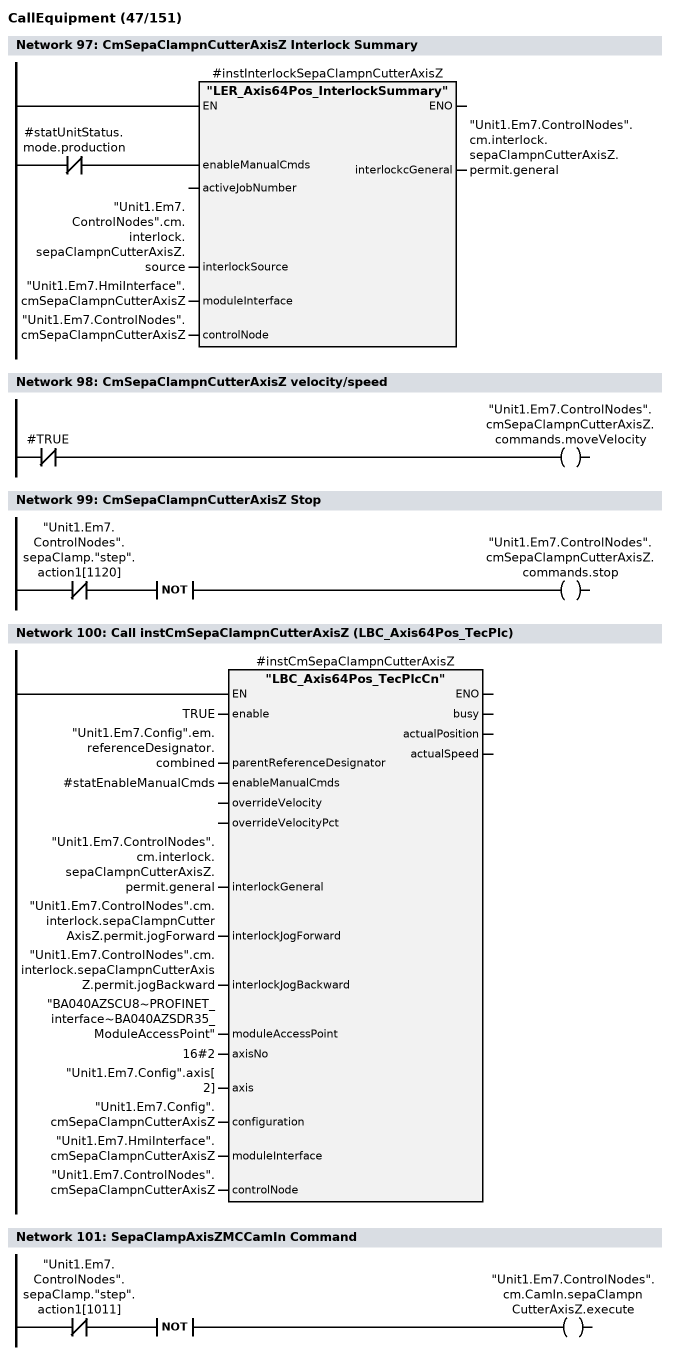
   RUNG wire#powerrail
      #instInterlockSepaClampnCutterAxisZ(enableManualCmds := wire#w1, activeJobNumber :=, interlockSource := "Unit1.Em7.ControlNodes".cm.interlock.sepaClampnCutterAxisZ.source, moduleInterface := "Unit1.Em7.HmiInterface".cmSepaClampnCutterAxisZ, controlNode := "Unit1.Em7.ControlNodes".cmSepaClampnCutterAxisZ, interlockcGeneral => "Unit1.Em7.ControlNodes".cm.interlock.sepaClampnCutterAxisZ.permit.general)
   END_RUNG
   RUNG wire#powerrail
      I_Contact( #statUnitStatus.mode.production )
   END_RUNG wire#w1
   // the same network as SCL:
   #instInterlockSepaClampnCutterAxisZ(enableManualCmds := NOT #statUnitStatus.mode.production,   // "LER_Axis64Pos_InterlockSummary"
                           interlockSource := "Unit1.Em7.ControlNodes".cm.interlock.sepaClampnCutterAxisZ.source,
                           moduleInterface := "Unit1.Em7.HmiInterface".cmSepaClampnCutterAxisZ,
                           controlNode := "Unit1.Em7.ControlNodes".cmSepaClampnCutterAxisZ,
                           interlockcGeneral => "Unit1.Em7.ControlNodes".cm.interlock.sepaClampnCutterAxisZ.permit.general);
END_REGION

REGION Network 98: CmSepaClampnCutterAxisZ velocity/speed
   RUNG wire#powerrail
      I_Contact( #TRUE )
      Coil( "Unit1.Em7.ControlNodes".cmSepaClampnCutterAxisZ.commands.moveVelocity )
   END_RUNG
   // the same network as SCL:
   "Unit1.Em7.ControlNodes".cmSepaClampnCutterAxisZ.commands.moveVelocity := NOT #TRUE;
END_REGION

REGION Network 99: CmSepaClampnCutterAxisZ Stop
   RUNG wire#powerrail
      I_Contact( "Unit1.Em7.ControlNodes".sepaClamp."step".action1[1120] )
      Not()
      Coil( "Unit1.Em7.ControlNodes".cmSepaClampnCutterAxisZ.commands.stop )
   END_RUNG
   // the same network as SCL:
   "Unit1.Em7.ControlNodes".cmSepaClampnCutterAxisZ.commands.stop := NOT (NOT "Unit1.Em7.ControlNodes".sepaClamp."step".action1[1120]);
END_REGION

REGION Network 100: Call instCmSepaClampnCutterAxisZ (LBC_Axis64Pos_TecPlc)
   RUNG wire#powerrail
      #instCmSepaClampnCutterAxisZ(enable := TRUE, parentReferenceDesignator := "Unit1.Em7.Config".em.referenceDesignator.combined, enableManualCmds := #statEnableManualCmds, overrideVelocity :=, overrideVelocityPct :=, interlockGeneral := "Unit1.Em7.ControlNodes".cm.interlock.sepaClampnCutterAxisZ.permit.general, interlockJogForward := "Unit1.Em7.ControlNodes".cm.interlock.sepaClampnCutterAxisZ.permit.jogForward, interlockJogBackward := "Unit1.Em7.ControlNodes".cm.interlock.sepaClampnCutterAxisZ.permit.jogBackward, moduleAccessPoint := "BA040AZSCU8~PROFINET_interface~BA040AZSDR35_ModuleAccessPoint", axisNo := 16#2, axis := "Unit1.Em7.Config".axis[2], configuration := "Unit1.Em7.Config".cmSepaClampnCutterAxisZ, moduleInterface := "Unit1.Em7.HmiInterface".cmSepaClampnCutterAxisZ, controlNode := "Unit1.Em7.ControlNodes".cmSepaClampnCutterAxisZ, busy =>, actualPosition =>, actualSpeed =>)
   END_RUNG
   // the same network as SCL:
   #instCmSepaClampnCutterAxisZ(enable := TRUE,   // "LBC_Axis64Pos_TecPlcCn"
                           parentReferenceDesignator := "Unit1.Em7.Config".em.referenceDesignator.combined,
                           enableManualCmds := #statEnableManualCmds,
                           interlockGeneral := "Unit1.Em7.ControlNodes".cm.interlock.sepaClampnCutterAxisZ.permit.general,
                           interlockJogForward := "Unit1.Em7.ControlNodes".cm.interlock.sepaClampnCutterAxisZ.permit.jogForward,
                           interlockJogBackward := "Unit1.Em7.ControlNodes".cm.interlock.sepaClampnCutterAxisZ.permit.jogBackward,
                           moduleAccessPoint := "BA040AZSCU8~PROFINET_interface~BA040AZSDR35_ModuleAccessPoint",
                           axisNo := 16#2,
                           axis := "Unit1.Em7.Config".axis[2],
                           configuration := "Unit1.Em7.Config".cmSepaClampnCutterAxisZ,
                           moduleInterface := "Unit1.Em7.HmiInterface".cmSepaClampnCutterAxisZ,
                           controlNode := "Unit1.Em7.ControlNodes".cmSepaClampnCutterAxisZ);
END_REGION

REGION Network 101: SepaClampAxisZMCCamIn Command
   RUNG wire#powerrail
      I_Contact( "Unit1.Em7.ControlNodes".sepaClamp."step".action1[1011] )
      Not()
      Coil( "Unit1.Em7.ControlNodes".cm.CamIn.sepaClampnCutterAxisZ.execute )
   END_RUNG
   // the same network as SCL:
   "Unit1.Em7.ControlNodes".cm.CamIn.sepaClampnCutterAxisZ.execute := NOT (NOT "Unit1.Em7.ControlNodes".sepaClamp."step".action1[1011]);
END_REGION

REGION Network 102: Call instSepaClampAxisZMCCamIn
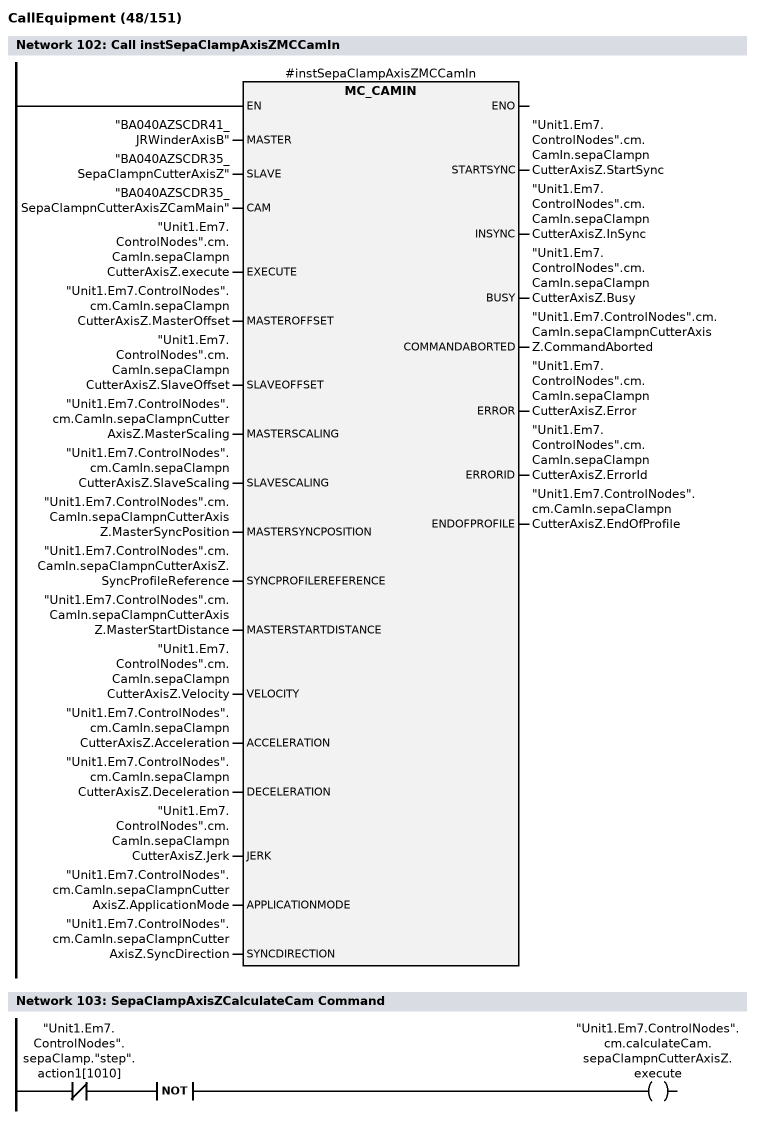
   RUNG wire#powerrail
      #instSepaClampAxisZMCCamIn.MC_CAMIN(Master := "BA040AZSCDR41_JRWinderAxisB", Slave := "BA040AZSCDR35_SepaClampnCutterAxisZ", Cam := "BA040AZSCDR35_SepaClampnCutterAxisZCamMain", Execute := "Unit1.Em7.ControlNodes".cm.CamIn.sepaClampnCutterAxisZ.execute, MasterOffset := "Unit1.Em7.ControlNodes".cm.CamIn.sepaClampnCutterAxisZ.MasterOffset, SlaveOffset := "Unit1.Em7.ControlNodes".cm.CamIn.sepaClampnCutterAxisZ.SlaveOffset, MasterScaling := "Unit1.Em7.ControlNodes".cm.CamIn.sepaClampnCutterAxisZ.MasterScaling, SlaveScaling := "Unit1.Em7.ControlNodes".cm.CamIn.sepaClampnCutterAxisZ.SlaveScaling, MasterSyncPosition := "Unit1.Em7.ControlNodes".cm.CamIn.sepaClampnCutterAxisZ.MasterSyncPosition, SyncProfileReference := "Unit1.Em7.ControlNodes".cm.CamIn.sepaClampnCutterAxisZ.SyncProfileReference, MasterStartDistance := "Unit1.Em7.ControlNodes".cm.CamIn.sepaClampnCutterAxisZ.MasterStartDistance, Velocity := "Unit1.Em7.ControlNodes".cm.CamIn.sepaClampnCutterAxisZ.Velocity, Acceleration := "Unit1.Em7.ControlNodes".cm.CamIn.sepaClampnCutterAxisZ.Acceleration, Deceleration := "Unit1.Em7.ControlNodes".cm.CamIn.sepaClampnCutterAxisZ.Deceleration, Jerk := "Unit1.Em7.ControlNodes".cm.CamIn.sepaClampnCutterAxisZ.Jerk, ApplicationMode := "Unit1.Em7.ControlNodes".cm.CamIn.sepaClampnCutterAxisZ.ApplicationMode, SyncDirection := "Unit1.Em7.ControlNodes".cm.CamIn.sepaClampnCutterAxisZ.SyncDirection, StartSync => "Unit1.Em7.ControlNodes".cm.CamIn.sepaClampnCutterAxisZ.StartSync, InSync => "Unit1.Em7.ControlNodes".cm.CamIn.sepaClampnCutterAxisZ.InSync, Busy => "Unit1.Em7.ControlNodes".cm.CamIn.sepaClampnCutterAxisZ.Busy, CommandAborted => "Unit1.Em7.ControlNodes".cm.CamIn.sepaClampnCutterAxisZ.CommandAborted, Error => "Unit1.Em7.ControlNodes".cm.CamIn.sepaClampnCutterAxisZ.Error, ErrorId => "Unit1.Em7.ControlNodes".cm.CamIn.sepaClampnCutterAxisZ.ErrorId, EndOfProfile => "Unit1.Em7.ControlNodes".cm.CamIn.sepaClampnCutterAxisZ.EndOfProfile)
   END_RUNG
   // the same network as SCL:
   #instSepaClampAxisZMCCamIn(Master := "BA040AZSCDR41_JRWinderAxisB",   // MC_CAMIN
                           Slave := "BA040AZSCDR35_SepaClampnCutterAxisZ",
                           Cam := "BA040AZSCDR35_SepaClampnCutterAxisZCamMain",
                           Execute := "Unit1.Em7.ControlNodes".cm.CamIn.sepaClampnCutterAxisZ.execute,
                           MasterOffset := "Unit1.Em7.ControlNodes".cm.CamIn.sepaClampnCutterAxisZ.MasterOffset,
                           SlaveOffset := "Unit1.Em7.ControlNodes".cm.CamIn.sepaClampnCutterAxisZ.SlaveOffset,
                           MasterScaling := "Unit1.Em7.ControlNodes".cm.CamIn.sepaClampnCutterAxisZ.MasterScaling,
                           SlaveScaling := "Unit1.Em7.ControlNodes".cm.CamIn.sepaClampnCutterAxisZ.SlaveScaling,
                           MasterSyncPosition := "Unit1.Em7.ControlNodes".cm.CamIn.sepaClampnCutterAxisZ.MasterSyncPosition,
                           SyncProfileReference := "Unit1.Em7.ControlNodes".cm.CamIn.sepaClampnCutterAxisZ.SyncProfileReference,
                           MasterStartDistance := "Unit1.Em7.ControlNodes".cm.CamIn.sepaClampnCutterAxisZ.MasterStartDistance,
                           Velocity := "Unit1.Em7.ControlNodes".cm.CamIn.sepaClampnCutterAxisZ.Velocity,
                           Acceleration := "Unit1.Em7.ControlNodes".cm.CamIn.sepaClampnCutterAxisZ.Acceleration,
                           Deceleration := "Unit1.Em7.ControlNodes".cm.CamIn.sepaClampnCutterAxisZ.Deceleration,
                           Jerk := "Unit1.Em7.ControlNodes".cm.CamIn.sepaClampnCutterAxisZ.Jerk,
                           ApplicationMode := "Unit1.Em7.ControlNodes".cm.CamIn.sepaClampnCutterAxisZ.ApplicationMode,
                           SyncDirection := "Unit1.Em7.ControlNodes".cm.CamIn.sepaClampnCutterAxisZ.SyncDirection,
                           StartSync => "Unit1.Em7.ControlNodes".cm.CamIn.sepaClampnCutterAxisZ.StartSync,
                           InSync => "Unit1.Em7.ControlNodes".cm.CamIn.sepaClampnCutterAxisZ.InSync,
                           Busy => "Unit1.Em7.ControlNodes".cm.CamIn.sepaClampnCutterAxisZ.Busy,
                           CommandAborted => "Unit1.Em7.ControlNodes".cm.CamIn.sepaClampnCutterAxisZ.CommandAborted,
                           Error => "Unit1.Em7.ControlNodes".cm.CamIn.sepaClampnCutterAxisZ.Error,
                           ErrorId => "Unit1.Em7.ControlNodes".cm.CamIn.sepaClampnCutterAxisZ.ErrorId,
                           EndOfProfile => "Unit1.Em7.ControlNodes".cm.CamIn.sepaClampnCutterAxisZ.EndOfProfile);
END_REGION

REGION Network 103: SepaClampAxisZCalculateCam Command
   RUNG wire#powerrail
      I_Contact( "Unit1.Em7.ControlNodes".sepaClamp."step".action1[1010] )
      Not()
      Coil( "Unit1.Em7.ControlNodes".cm.calculateCam.sepaClampnCutterAxisZ.execute )
   END_RUNG
   // the same network as SCL:
   "Unit1.Em7.ControlNodes".cm.calculateCam.sepaClampnCutterAxisZ.execute := NOT (NOT "Unit1.Em7.ControlNodes".sepaClamp."step".action1[1010]);
END_REGION

REGION Network 104: Call instSepaClampAxisZCalculateCam
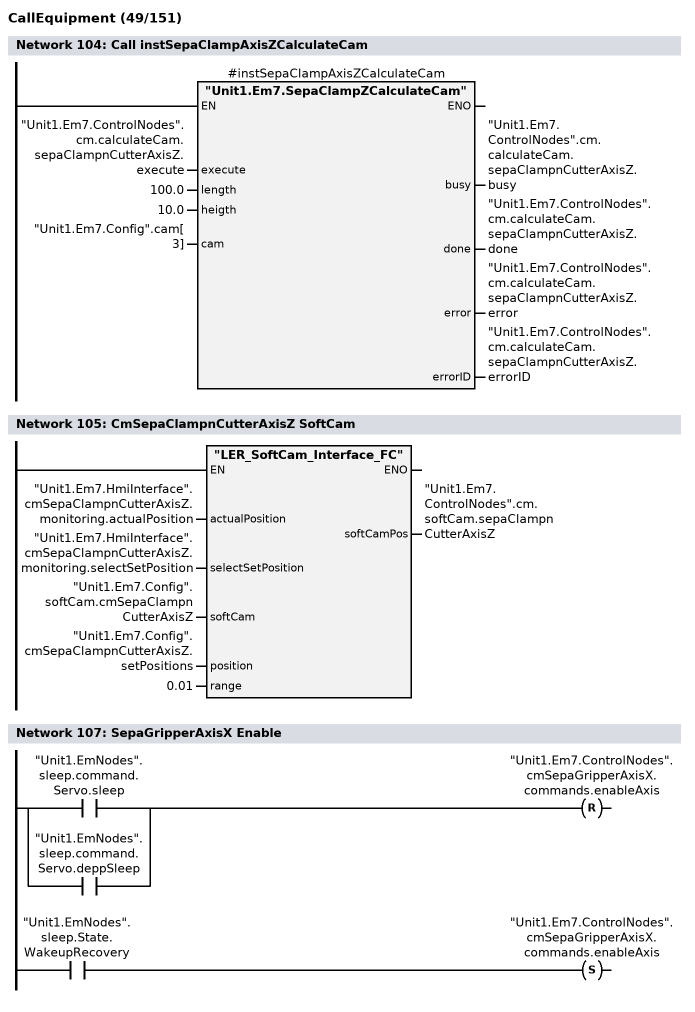
   RUNG wire#powerrail
      #instSepaClampAxisZCalculateCam(execute := "Unit1.Em7.ControlNodes".cm.calculateCam.sepaClampnCutterAxisZ.execute, length := 100.0, heigth := 10.0, cam := "Unit1.Em7.Config".cam[3], busy => "Unit1.Em7.ControlNodes".cm.calculateCam.sepaClampnCutterAxisZ.busy, done => "Unit1.Em7.ControlNodes".cm.calculateCam.sepaClampnCutterAxisZ.done, error => "Unit1.Em7.ControlNodes".cm.calculateCam.sepaClampnCutterAxisZ.error, errorID => "Unit1.Em7.ControlNodes".cm.calculateCam.sepaClampnCutterAxisZ.errorID)
   END_RUNG
   // the same network as SCL:
   #instSepaClampAxisZCalculateCam(execute := "Unit1.Em7.ControlNodes".cm.calculateCam.sepaClampnCutterAxisZ.execute,   // "Unit1.Em7.SepaClampZCalculateCam"
                           length := 100.0,
                           heigth := 10.0,
                           cam := "Unit1.Em7.Config".cam[3],
                           busy => "Unit1.Em7.ControlNodes".cm.calculateCam.sepaClampnCutterAxisZ.busy,
                           done => "Unit1.Em7.ControlNodes".cm.calculateCam.sepaClampnCutterAxisZ.done,
                           error => "Unit1.Em7.ControlNodes".cm.calculateCam.sepaClampnCutterAxisZ.error,
                           errorID => "Unit1.Em7.ControlNodes".cm.calculateCam.sepaClampnCutterAxisZ.errorID);
END_REGION

REGION Network 105: CmSepaClampnCutterAxisZ SoftCam
   RUNG wire#powerrail
      "LER_SoftCam_Interface_FC"(actualPosition := "Unit1.Em7.HmiInterface".cmSepaClampnCutterAxisZ.monitoring.actualPosition, selectSetPosition := "Unit1.Em7.HmiInterface".cmSepaClampnCutterAxisZ.monitoring.selectSetPosition, softCam := "Unit1.Em7.Config".softCam.cmSepaClampnCutterAxisZ, position := "Unit1.Em7.Config".cmSepaClampnCutterAxisZ.setPositions, range := 0.01, softCamPos => "Unit1.Em7.ControlNodes".cm.softCam.sepaClampnCutterAxisZ)
   END_RUNG
   // the same network as SCL:
   "LER_SoftCam_Interface_FC"(actualPosition := "Unit1.Em7.HmiInterface".cmSepaClampnCutterAxisZ.monitoring.actualPosition,
                           selectSetPosition := "Unit1.Em7.HmiInterface".cmSepaClampnCutterAxisZ.monitoring.selectSetPosition,
                           softCam := "Unit1.Em7.Config".softCam.cmSepaClampnCutterAxisZ,
                           position := "Unit1.Em7.Config".cmSepaClampnCutterAxisZ.setPositions,
                           range := 0.01,
                           softCamPos => "Unit1.Em7.ControlNodes".cm.softCam.sepaClampnCutterAxisZ);
END_REGION

REGION Network 107: SepaGripperAxisX Enable
   RUNG wire#powerrail
      Contact( "Unit1.EmNodes".sleep.command.Servo.sleep )
      wire#w1
      R_Coil( "Unit1.Em7.ControlNodes".cmSepaGripperAxisX.commands.enableAxis )
   END_RUNG
   RUNG wire#powerrail
      Contact( "Unit1.EmNodes".sleep.command.Servo.deppSleep )
   END_RUNG wire#w1
   RUNG wire#powerrail
      Contact( "Unit1.EmNodes".sleep.State.WakeupRecovery )
      S_Coil( "Unit1.Em7.ControlNodes".cmSepaGripperAxisX.commands.enableAxis )
   END_RUNG
   // the same network as SCL:
   IF "Unit1.EmNodes".sleep.command.Servo.sleep OR "Unit1.EmNodes".sleep.command.Servo.deppSleep THEN
       "Unit1.Em7.ControlNodes".cmSepaGripperAxisX.commands.enableAxis := FALSE;
   END_IF;
   IF "Unit1.EmNodes".sleep.State.WakeupRecovery THEN
       "Unit1.Em7.ControlNodes".cmSepaGripperAxisX.commands.enableAxis := TRUE;
   END_IF;
END_REGION

REGION Network 108: CmSepaGripperAxisX Position Absolute Home
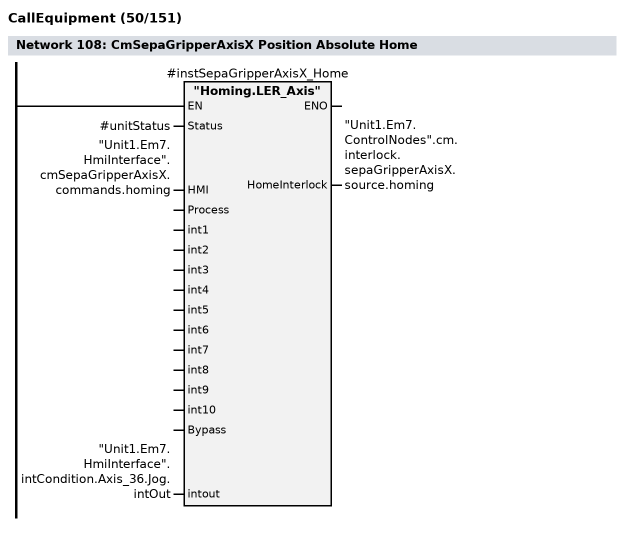
   RUNG wire#powerrail
      #instSepaGripperAxisX_Home(Status := #unitStatus, HMI := "Unit1.Em7.HmiInterface".cmSepaGripperAxisX.commands.homing, Process :=, int1 :=, int2 :=, int3 :=, int4 :=, int5 :=, int6 :=, int7 :=, int8 :=, int9 :=, int10 :=, Bypass :=, intout := "Unit1.Em7.HmiInterface".intCondition.Axis_36.Jog.intOut, HomeInterlock => "Unit1.Em7.ControlNodes".cm.interlock.sepaGripperAxisX.source.homing)
   END_RUNG
   // the same network as SCL:
   #instSepaGripperAxisX_Home(Status := #unitStatus,   // "Homing.LER_Axis"
                           HMI := "Unit1.Em7.HmiInterface".cmSepaGripperAxisX.commands.homing,
                           intout := "Unit1.Em7.HmiInterface".intCondition.Axis_36.Jog.intOut,
                           HomeInterlock => "Unit1.Em7.ControlNodes".cm.interlock.sepaGripperAxisX.source.homing);
END_REGION

REGION Network 109: CmSepaGripperAxisX Position Absolute Jog
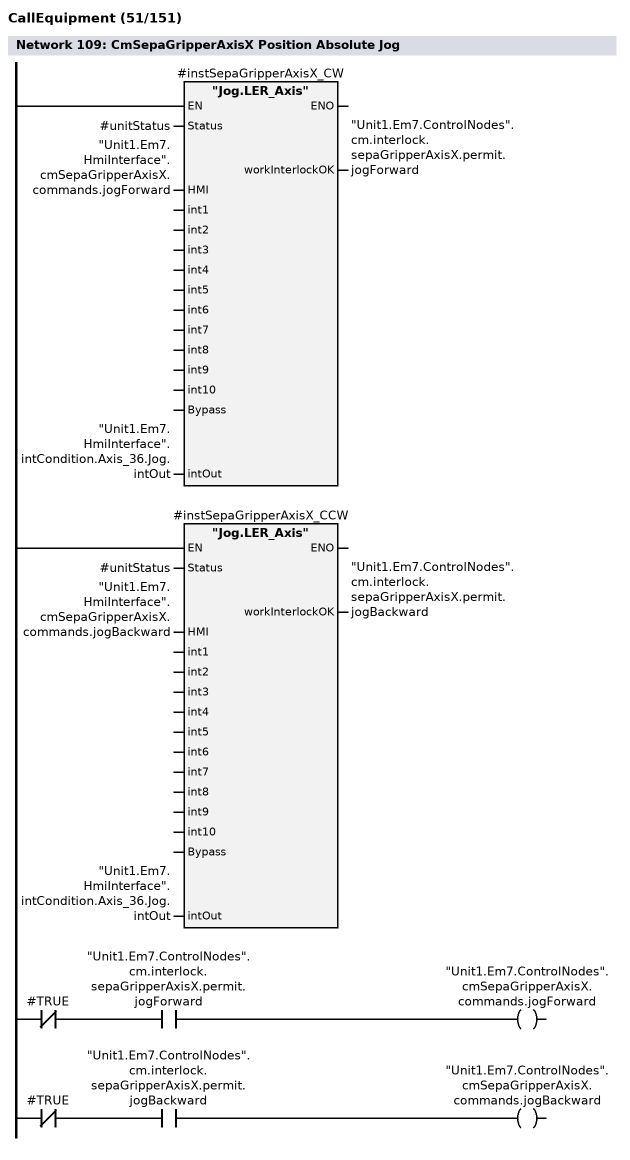
   RUNG wire#powerrail
      #instSepaGripperAxisX_CW(Status := #unitStatus, HMI := "Unit1.Em7.HmiInterface".cmSepaGripperAxisX.commands.jogForward, int1 :=, int2 :=, int3 :=, int4 :=, int5 :=, int6 :=, int7 :=, int8 :=, int9 :=, int10 :=, Bypass :=, intOut := "Unit1.Em7.HmiInterface".intCondition.Axis_36.Jog.intOut, workInterlockOK => "Unit1.Em7.ControlNodes".cm.interlock.sepaGripperAxisX.permit.jogForward)
   END_RUNG
   RUNG wire#powerrail
      #instSepaGripperAxisX_CCW(Status := #unitStatus, HMI := "Unit1.Em7.HmiInterface".cmSepaGripperAxisX.commands.jogBackward, int1 :=, int2 :=, int3 :=, int4 :=, int5 :=, int6 :=, int7 :=, int8 :=, int9 :=, int10 :=, Bypass :=, intOut := "Unit1.Em7.HmiInterface".intCondition.Axis_36.Jog.intOut, workInterlockOK => "Unit1.Em7.ControlNodes".cm.interlock.sepaGripperAxisX.permit.jogBackward)
   END_RUNG
   RUNG wire#powerrail
      I_Contact( #TRUE )
      Contact( "Unit1.Em7.ControlNodes".cm.interlock.sepaGripperAxisX.permit.jogForward )
      Coil( "Unit1.Em7.ControlNodes".cmSepaGripperAxisX.commands.jogForward )
   END_RUNG
   RUNG wire#powerrail
      I_Contact( #TRUE )
      Contact( "Unit1.Em7.ControlNodes".cm.interlock.sepaGripperAxisX.permit.jogBackward )
      Coil( "Unit1.Em7.ControlNodes".cmSepaGripperAxisX.commands.jogBackward )
   END_RUNG
   // the same network as SCL:
   #instSepaGripperAxisX_CW(Status := #unitStatus,   // "Jog.LER_Axis"
                           HMI := "Unit1.Em7.HmiInterface".cmSepaGripperAxisX.commands.jogForward,
                           intOut := "Unit1.Em7.HmiInterface".intCondition.Axis_36.Jog.intOut,
                           workInterlockOK => "Unit1.Em7.ControlNodes".cm.interlock.sepaGripperAxisX.permit.jogForward);
   #instSepaGripperAxisX_CCW(Status := #unitStatus,   // "Jog.LER_Axis"
                           HMI := "Unit1.Em7.HmiInterface".cmSepaGripperAxisX.commands.jogBackward,
                           intOut := "Unit1.Em7.HmiInterface".intCondition.Axis_36.Jog.intOut,
                           workInterlockOK => "Unit1.Em7.ControlNodes".cm.interlock.sepaGripperAxisX.permit.jogBackward);
   "Unit1.Em7.ControlNodes".cmSepaGripperAxisX.commands.jogForward := NOT #TRUE AND "Unit1.Em7.ControlNodes".cm.interlock.sepaGripperAxisX.permit.jogForward;
   "Unit1.Em7.ControlNodes".cmSepaGripperAxisX.commands.jogBackward := NOT #TRUE AND "Unit1.Em7.ControlNodes".cm.interlock.sepaGripperAxisX.permit.jogBackward;
END_REGION

REGION Network 110: CmSepaGripperAxisX Position Absolute Position0
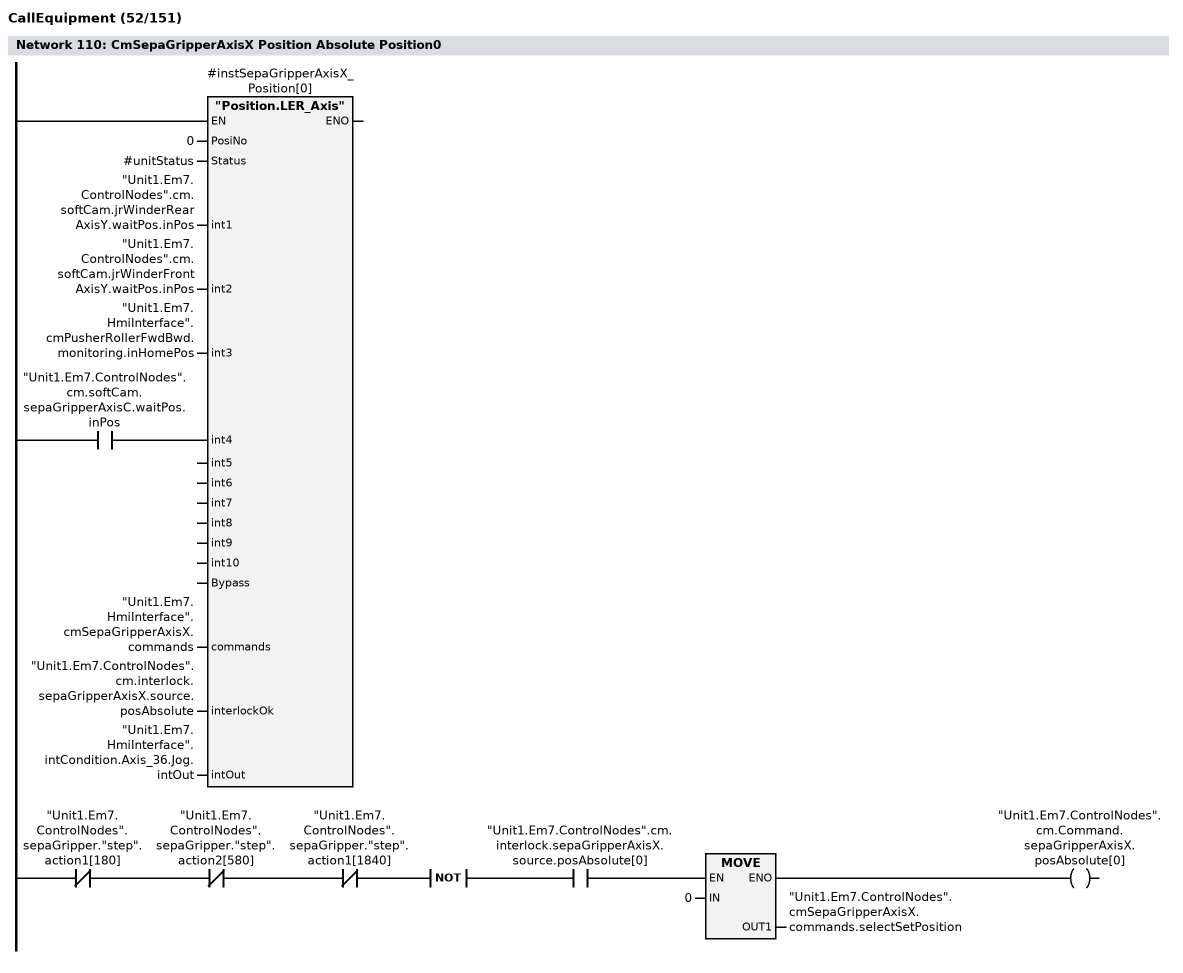
   RUNG wire#powerrail
      #instSepaGripperAxisX_Position[0](int4 := wire#w1, PosiNo := 0, Status := #unitStatus, int1 := "Unit1.Em7.ControlNodes".cm.softCam.jrWinderRearAxisY.waitPos.inPos, int2 := "Unit1.Em7.ControlNodes".cm.softCam.jrWinderFrontAxisY.waitPos.inPos, int3 := "Unit1.Em7.HmiInterface".cmPusherRollerFwdBwd.monitoring.inHomePos, int5 :=, int6 :=, int7 :=, int8 :=, int9 :=, int10 :=, Bypass :=, commands := "Unit1.Em7.HmiInterface".cmSepaGripperAxisX.commands, interlockOk := "Unit1.Em7.ControlNodes".cm.interlock.sepaGripperAxisX.source.posAbsolute, intOut := "Unit1.Em7.HmiInterface".intCondition.Axis_36.Jog.intOut)
   END_RUNG
   RUNG wire#powerrail
      Contact( "Unit1.Em7.ControlNodes".cm.softCam.sepaGripperAxisC.waitPos.inPos )
   END_RUNG wire#w1
   RUNG wire#powerrail
      I_Contact( "Unit1.Em7.ControlNodes".sepaGripper."step".action1[180] )
      I_Contact( "Unit1.Em7.ControlNodes".sepaGripper."step".action2[580] )
      I_Contact( "Unit1.Em7.ControlNodes".sepaGripper."step".action1[1840] )
      Not()
      Contact( "Unit1.Em7.ControlNodes".cm.interlock.sepaGripperAxisX.source.posAbsolute[0] )
      Move(in := 0, out1 => "Unit1.Em7.ControlNodes".cmSepaGripperAxisX.commands.selectSetPosition)
      Coil( "Unit1.Em7.ControlNodes".cm.Command.sepaGripperAxisX.posAbsolute[0] )
   END_RUNG
   // the same network as SCL:
   #instSepaGripperAxisX_Position[0](PosiNo := 0,   // "Position.LER_Axis"
                           Status := #unitStatus,
                           int1 := "Unit1.Em7.ControlNodes".cm.softCam.jrWinderRearAxisY.waitPos.inPos,
                           int2 := "Unit1.Em7.ControlNodes".cm.softCam.jrWinderFrontAxisY.waitPos.inPos,
                           int3 := "Unit1.Em7.HmiInterface".cmPusherRollerFwdBwd.monitoring.inHomePos,
                           int4 := "Unit1.Em7.ControlNodes".cm.softCam.sepaGripperAxisC.waitPos.inPos,
                           commands := "Unit1.Em7.HmiInterface".cmSepaGripperAxisX.commands,
                           interlockOk := "Unit1.Em7.ControlNodes".cm.interlock.sepaGripperAxisX.source.posAbsolute,
                           intOut := "Unit1.Em7.HmiInterface".intCondition.Axis_36.Jog.intOut);
   #_w1 := NOT (NOT "Unit1.Em7.ControlNodes".sepaGripper."step".action1[180] AND NOT "Unit1.Em7.ControlNodes".sepaGripper."step".action2[580] AND NOT "Unit1.Em7.ControlNodes".sepaGripper."step".action1[1840]) AND "Unit1.Em7.ControlNodes".cm.interlock.sepaGripperAxisX.source.posAbsolute[0];
   IF #_w1 THEN "Unit1.Em7.ControlNodes".cmSepaGripperAxisX.commands.selectSetPosition := 0; END_IF;
   "Unit1.Em7.ControlNodes".cm.Command.sepaGripperAxisX.posAbsolute[0] := #_w1;
END_REGION

REGION Network 111: CmSepaGripperAxisX Position Absolute Position1
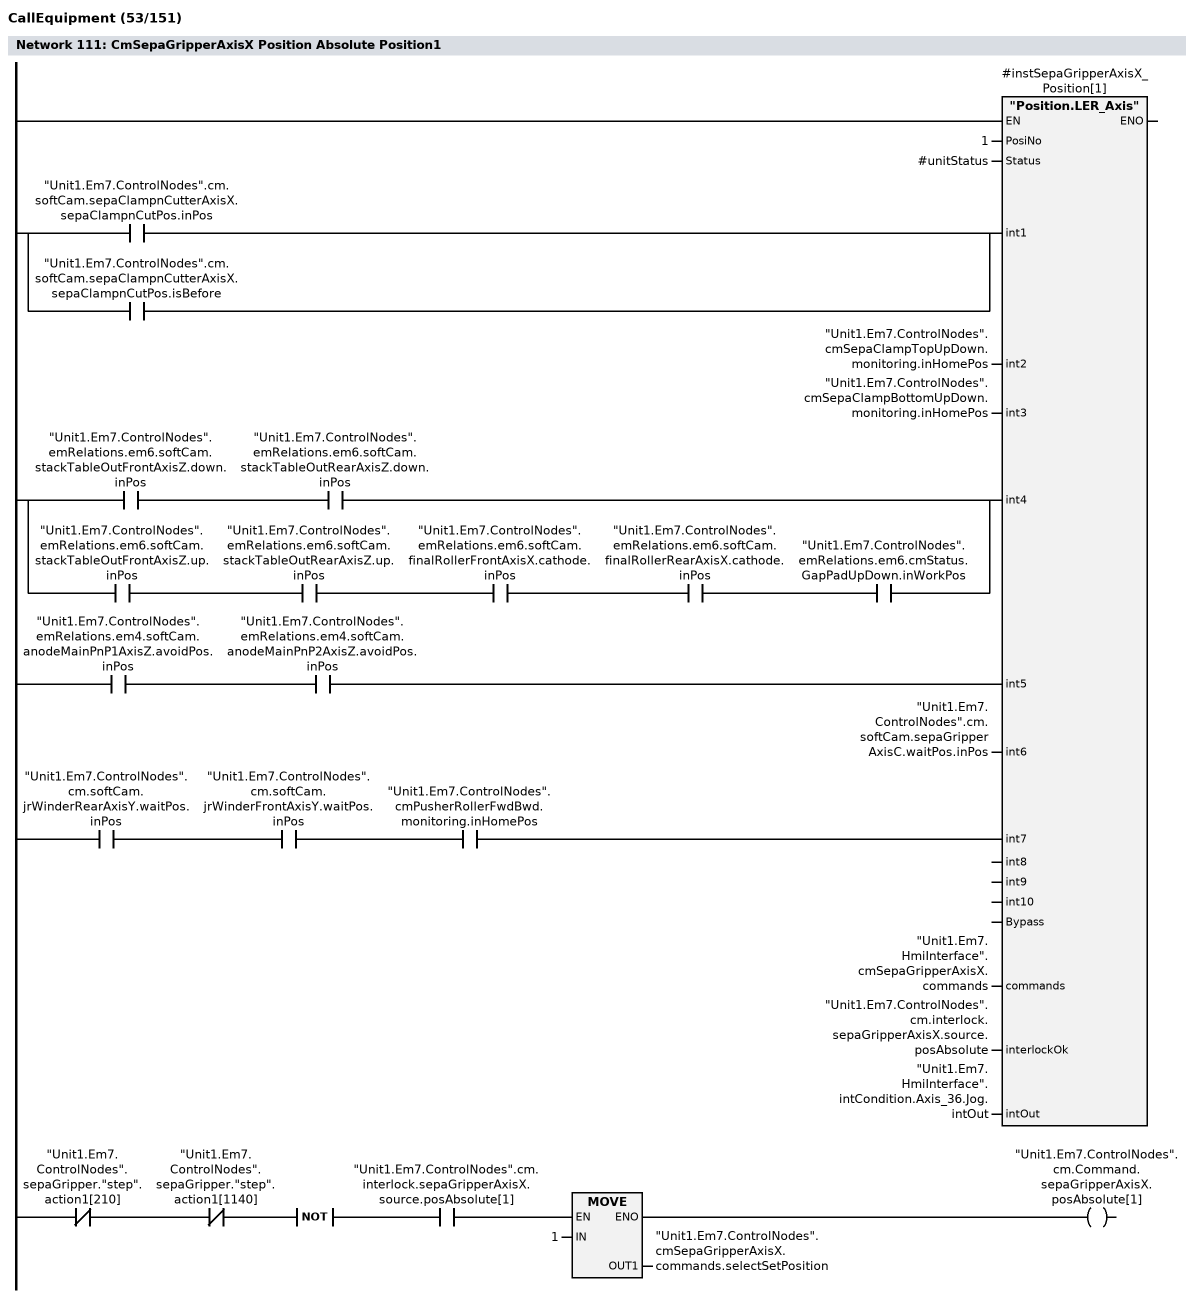
   RUNG wire#powerrail
      #instSepaGripperAxisX_Position[1](int1 := wire#w1, int4 := wire#w2, int5 := wire#w3, int7 := wire#w4, PosiNo := 1, Status := #unitStatus, int2 := "Unit1.Em7.ControlNodes".cmSepaClampTopUpDown.monitoring.inHomePos, int3 := "Unit1.Em7.ControlNodes".cmSepaClampBottomUpDown.monitoring.inHomePos, int6 := "Unit1.Em7.ControlNodes".cm.softCam.sepaGripperAxisC.waitPos.inPos, int8 :=, int9 :=, int10 :=, Bypass :=, commands := "Unit1.Em7.HmiInterface".cmSepaGripperAxisX.commands, interlockOk := "Unit1.Em7.ControlNodes".cm.interlock.sepaGripperAxisX.source.posAbsolute, intOut := "Unit1.Em7.HmiInterface".intCondition.Axis_36.Jog.intOut)
   END_RUNG
   RUNG wire#powerrail
      Contact( "Unit1.Em7.ControlNodes".cm.softCam.sepaClampnCutterAxisX.sepaClampnCutPos.inPos )
   END_RUNG wire#w1
   RUNG wire#powerrail
      Contact( "Unit1.Em7.ControlNodes".cm.softCam.sepaClampnCutterAxisX.sepaClampnCutPos.isBefore )
   END_RUNG wire#w1
   RUNG wire#powerrail
      Contact( "Unit1.Em7.ControlNodes".emRelations.em6.softCam.stackTableOutFrontAxisZ.down.inPos )
      Contact( "Unit1.Em7.ControlNodes".emRelations.em6.softCam.stackTableOutRearAxisZ.down.inPos )
   END_RUNG wire#w2
   RUNG wire#powerrail
      Contact( "Unit1.Em7.ControlNodes".emRelations.em6.softCam.stackTableOutFrontAxisZ.up.inPos )
      Contact( "Unit1.Em7.ControlNodes".emRelations.em6.softCam.stackTableOutRearAxisZ.up.inPos )
      Contact( "Unit1.Em7.ControlNodes".emRelations.em6.softCam.finalRollerFrontAxisX.cathode.inPos )
      Contact( "Unit1.Em7.ControlNodes".emRelations.em6.softCam.finalRollerRearAxisX.cathode.inPos )
      Contact( "Unit1.Em7.ControlNodes".emRelations.em6.cmStatus.GapPadUpDown.inWorkPos )
   END_RUNG wire#w2
   RUNG wire#powerrail
      Contact( "Unit1.Em7.ControlNodes".emRelations.em4.softCam.anodeMainPnP1AxisZ.avoidPos.inPos )
      Contact( "Unit1.Em7.ControlNodes".emRelations.em4.softCam.anodeMainPnP2AxisZ.avoidPos.inPos )
   END_RUNG wire#w3
   RUNG wire#powerrail
      Contact( "Unit1.Em7.ControlNodes".cm.softCam.jrWinderRearAxisY.waitPos.inPos )
      Contact( "Unit1.Em7.ControlNodes".cm.softCam.jrWinderFrontAxisY.waitPos.inPos )
      Contact( "Unit1.Em7.ControlNodes".cmPusherRollerFwdBwd.monitoring.inHomePos )
   END_RUNG wire#w4
   RUNG wire#powerrail
      I_Contact( "Unit1.Em7.ControlNodes".sepaGripper."step".action1[210] )
      I_Contact( "Unit1.Em7.ControlNodes".sepaGripper."step".action1[1140] )
      Not()
      Contact( "Unit1.Em7.ControlNodes".cm.interlock.sepaGripperAxisX.source.posAbsolute[1] )
      Move(in := 1, out1 => "Unit1.Em7.ControlNodes".cmSepaGripperAxisX.commands.selectSetPosition)
      Coil( "Unit1.Em7.ControlNodes".cm.Command.sepaGripperAxisX.posAbsolute[1] )
   END_RUNG
   // the same network as SCL:
   #instSepaGripperAxisX_Position[1](PosiNo := 1,   // "Position.LER_Axis"
                           Status := #unitStatus,
                           int1 := "Unit1.Em7.ControlNodes".cm.softCam.sepaClampnCutterAxisX.sepaClampnCutPos.inPos OR "Unit1.Em7.ControlNodes".cm.softCam.sepaClampnCutterAxisX.sepaClampnCutPos.isBefore,
                           int2 := "Unit1.Em7.ControlNodes".cmSepaClampTopUpDown.monitoring.inHomePos,
                           int3 := "Unit1.Em7.ControlNodes".cmSepaClampBottomUpDown.monitoring.inHomePos,
                           int4 := ("Unit1.Em7.ControlNodes".emRelations.em6.softCam.stackTableOutFrontAxisZ.down.inPos AND "Unit1.Em7.ControlNodes".emRelations.em6.softCam.stackTableOutRearAxisZ.down.inPos) OR ("Unit1.Em7.ControlNodes".emRelations.em6.softCam.stackTableOutFrontAxisZ.up.inPos AND "Unit1.Em7.ControlNodes".emRelations.em6.softCam.stackTableOutRearAxisZ.up.inPos AND "Unit1.Em7.ControlNodes".emRelations.em6.softCam.finalRollerFrontAxisX.cathode.inPos AND "Unit1.Em7.ControlNodes".emRelations.em6.softCam.finalRollerRearAxisX.cathode.inPos AND "Unit1.Em7.ControlNodes".emRelations.em6.cmStatus.GapPadUpDown.inWorkPos),
                           int5 := "Unit1.Em7.ControlNodes".emRelations.em4.softCam.anodeMainPnP1AxisZ.avoidPos.inPos AND "Unit1.Em7.ControlNodes".emRelations.em4.softCam.anodeMainPnP2AxisZ.avoidPos.inPos,
                           int6 := "Unit1.Em7.ControlNodes".cm.softCam.sepaGripperAxisC.waitPos.inPos,
                           int7 := "Unit1.Em7.ControlNodes".cm.softCam.jrWinderRearAxisY.waitPos.inPos AND "Unit1.Em7.ControlNodes".cm.softCam.jrWinderFrontAxisY.waitPos.inPos AND "Unit1.Em7.ControlNodes".cmPusherRollerFwdBwd.monitoring.inHomePos,
                           commands := "Unit1.Em7.HmiInterface".cmSepaGripperAxisX.commands,
                           interlockOk := "Unit1.Em7.ControlNodes".cm.interlock.sepaGripperAxisX.source.posAbsolute,
                           intOut := "Unit1.Em7.HmiInterface".intCondition.Axis_36.Jog.intOut);
   #_w1 := NOT (NOT "Unit1.Em7.ControlNodes".sepaGripper."step".action1[210] AND NOT "Unit1.Em7.ControlNodes".sepaGripper."step".action1[1140]) AND "Unit1.Em7.ControlNodes".cm.interlock.sepaGripperAxisX.source.posAbsolute[1];
   IF #_w1 THEN "Unit1.Em7.ControlNodes".cmSepaGripperAxisX.commands.selectSetPosition := 1; END_IF;
   "Unit1.Em7.ControlNodes".cm.Command.sepaGripperAxisX.posAbsolute[1] := #_w1;
END_REGION

REGION Network 112: CmSepaGripperAxisX Position Absolute Position2
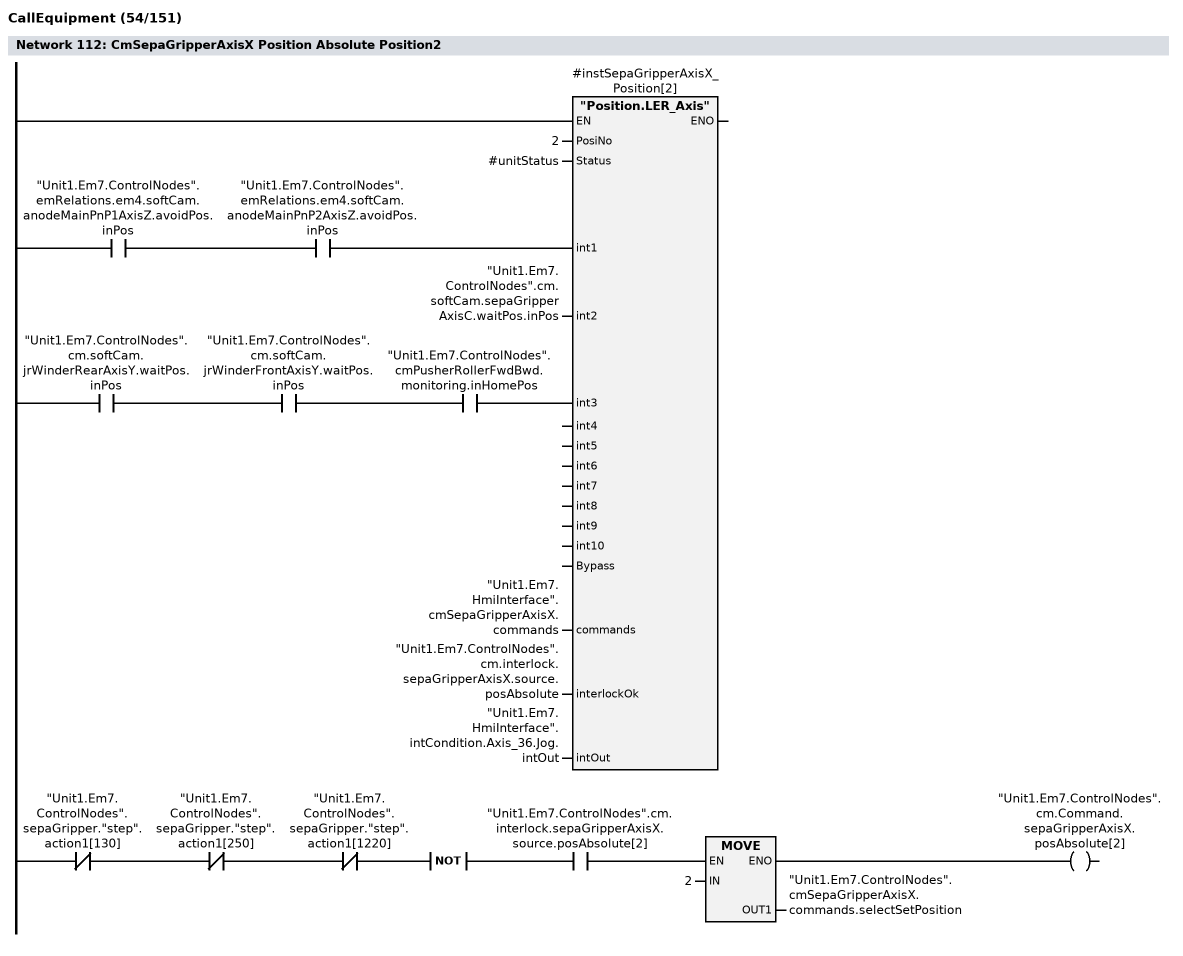
   RUNG wire#powerrail
      #instSepaGripperAxisX_Position[2](int1 := wire#w1, int3 := wire#w2, PosiNo := 2, Status := #unitStatus, int2 := "Unit1.Em7.ControlNodes".cm.softCam.sepaGripperAxisC.waitPos.inPos, int4 :=, int5 :=, int6 :=, int7 :=, int8 :=, int9 :=, int10 :=, Bypass :=, commands := "Unit1.Em7.HmiInterface".cmSepaGripperAxisX.commands, interlockOk := "Unit1.Em7.ControlNodes".cm.interlock.sepaGripperAxisX.source.posAbsolute, intOut := "Unit1.Em7.HmiInterface".intCondition.Axis_36.Jog.intOut)
   END_RUNG
   RUNG wire#powerrail
      Contact( "Unit1.Em7.ControlNodes".emRelations.em4.softCam.anodeMainPnP1AxisZ.avoidPos.inPos )
      Contact( "Unit1.Em7.ControlNodes".emRelations.em4.softCam.anodeMainPnP2AxisZ.avoidPos.inPos )
   END_RUNG wire#w1
   RUNG wire#powerrail
      Contact( "Unit1.Em7.ControlNodes".cm.softCam.jrWinderRearAxisY.waitPos.inPos )
      Contact( "Unit1.Em7.ControlNodes".cm.softCam.jrWinderFrontAxisY.waitPos.inPos )
      Contact( "Unit1.Em7.ControlNodes".cmPusherRollerFwdBwd.monitoring.inHomePos )
   END_RUNG wire#w2
   RUNG wire#powerrail
      I_Contact( "Unit1.Em7.ControlNodes".sepaGripper."step".action1[130] )
      I_Contact( "Unit1.Em7.ControlNodes".sepaGripper."step".action1[250] )
      I_Contact( "Unit1.Em7.ControlNodes".sepaGripper."step".action1[1220] )
      Not()
      Contact( "Unit1.Em7.ControlNodes".cm.interlock.sepaGripperAxisX.source.posAbsolute[2] )
      Move(in := 2, out1 => "Unit1.Em7.ControlNodes".cmSepaGripperAxisX.commands.selectSetPosition)
      Coil( "Unit1.Em7.ControlNodes".cm.Command.sepaGripperAxisX.posAbsolute[2] )
   END_RUNG
   // the same network as SCL:
   #instSepaGripperAxisX_Position[2](PosiNo := 2,   // "Position.LER_Axis"
                           Status := #unitStatus,
                           int1 := "Unit1.Em7.ControlNodes".emRelations.em4.softCam.anodeMainPnP1AxisZ.avoidPos.inPos AND "Unit1.Em7.ControlNodes".emRelations.em4.softCam.anodeMainPnP2AxisZ.avoidPos.inPos,
                           int2 := "Unit1.Em7.ControlNodes".cm.softCam.sepaGripperAxisC.waitPos.inPos,
                           int3 := "Unit1.Em7.ControlNodes".cm.softCam.jrWinderRearAxisY.waitPos.inPos AND "Unit1.Em7.ControlNodes".cm.softCam.jrWinderFrontAxisY.waitPos.inPos AND "Unit1.Em7.ControlNodes".cmPusherRollerFwdBwd.monitoring.inHomePos,
                           commands := "Unit1.Em7.HmiInterface".cmSepaGripperAxisX.commands,
                           interlockOk := "Unit1.Em7.ControlNodes".cm.interlock.sepaGripperAxisX.source.posAbsolute,
                           intOut := "Unit1.Em7.HmiInterface".intCondition.Axis_36.Jog.intOut);
   #_w1 := NOT (NOT "Unit1.Em7.ControlNodes".sepaGripper."step".action1[130] AND NOT "Unit1.Em7.ControlNodes".sepaGripper."step".action1[250] AND NOT "Unit1.Em7.ControlNodes".sepaGripper."step".action1[1220]) AND "Unit1.Em7.ControlNodes".cm.interlock.sepaGripperAxisX.source.posAbsolute[2];
   IF #_w1 THEN "Unit1.Em7.ControlNodes".cmSepaGripperAxisX.commands.selectSetPosition := 2; END_IF;
   "Unit1.Em7.ControlNodes".cm.Command.sepaGripperAxisX.posAbsolute[2] := #_w1;
END_REGION

REGION Network 113: CmSepaGripperAxisX Position Absolute Position3
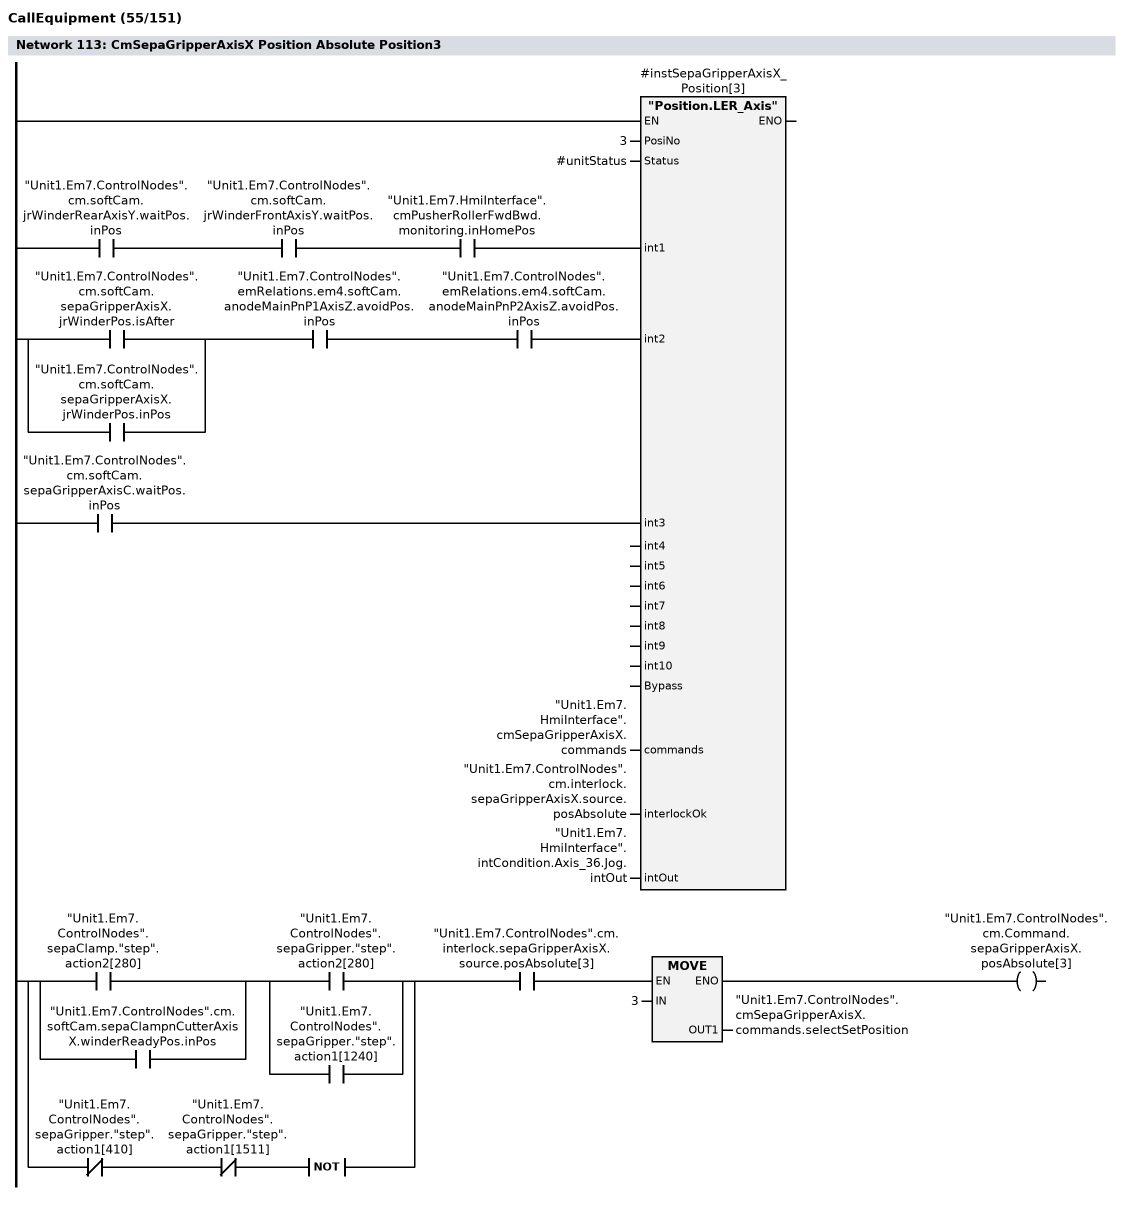
   RUNG wire#powerrail
      #instSepaGripperAxisX_Position[3](int1 := wire#w1, int2 := wire#w3, int3 := wire#w4, PosiNo := 3, Status := #unitStatus, int4 :=, int5 :=, int6 :=, int7 :=, int8 :=, int9 :=, int10 :=, Bypass :=, commands := "Unit1.Em7.HmiInterface".cmSepaGripperAxisX.commands, interlockOk := "Unit1.Em7.ControlNodes".cm.interlock.sepaGripperAxisX.source.posAbsolute, intOut := "Unit1.Em7.HmiInterface".intCondition.Axis_36.Jog.intOut)
   END_RUNG
   RUNG wire#powerrail
      Contact( "Unit1.Em7.ControlNodes".cm.softCam.jrWinderRearAxisY.waitPos.inPos )
      Contact( "Unit1.Em7.ControlNodes".cm.softCam.jrWinderFrontAxisY.waitPos.inPos )
      Contact( "Unit1.Em7.HmiInterface".cmPusherRollerFwdBwd.monitoring.inHomePos )
   END_RUNG wire#w1
   RUNG wire#powerrail
      Contact( "Unit1.Em7.ControlNodes".cm.softCam.sepaGripperAxisX.jrWinderPos.isAfter )
      wire#w2
      Contact( "Unit1.Em7.ControlNodes".emRelations.em4.softCam.anodeMainPnP1AxisZ.avoidPos.inPos )
      Contact( "Unit1.Em7.ControlNodes".emRelations.em4.softCam.anodeMainPnP2AxisZ.avoidPos.inPos )
   END_RUNG wire#w3
   RUNG wire#powerrail
      Contact( "Unit1.Em7.ControlNodes".cm.softCam.sepaGripperAxisX.jrWinderPos.inPos )
   END_RUNG wire#w2
   RUNG wire#powerrail
      Contact( "Unit1.Em7.ControlNodes".cm.softCam.sepaGripperAxisC.waitPos.inPos )
   END_RUNG wire#w4
   RUNG wire#powerrail
      Contact( "Unit1.Em7.ControlNodes".sepaClamp."step".action2[280] )
      wire#w5
      Contact( "Unit1.Em7.ControlNodes".sepaGripper."step".action2[280] )
      wire#w6
      Contact( "Unit1.Em7.ControlNodes".cm.interlock.sepaGripperAxisX.source.posAbsolute[3] )
      Move(in := 3, out1 => "Unit1.Em7.ControlNodes".cmSepaGripperAxisX.commands.selectSetPosition)
      Coil( "Unit1.Em7.ControlNodes".cm.Command.sepaGripperAxisX.posAbsolute[3] )
   END_RUNG
   RUNG wire#powerrail
      Contact( "Unit1.Em7.ControlNodes".cm.softCam.sepaClampnCutterAxisX.winderReadyPos.inPos )
   END_RUNG wire#w5
   RUNG wire#w5
      Contact( "Unit1.Em7.ControlNodes".sepaGripper."step".action1[1240] )
   END_RUNG wire#w6
   RUNG wire#powerrail
      I_Contact( "Unit1.Em7.ControlNodes".sepaGripper."step".action1[410] )
      I_Contact( "Unit1.Em7.ControlNodes".sepaGripper."step".action1[1511] )
      Not()
   END_RUNG wire#w6
   // the same network as SCL:
   #instSepaGripperAxisX_Position[3](PosiNo := 3,   // "Position.LER_Axis"
                           Status := #unitStatus,
                           int1 := "Unit1.Em7.ControlNodes".cm.softCam.jrWinderRearAxisY.waitPos.inPos AND "Unit1.Em7.ControlNodes".cm.softCam.jrWinderFrontAxisY.waitPos.inPos AND "Unit1.Em7.HmiInterface".cmPusherRollerFwdBwd.monitoring.inHomePos,
                           int2 := ("Unit1.Em7.ControlNodes".cm.softCam.sepaGripperAxisX.jrWinderPos.isAfter OR "Unit1.Em7.ControlNodes".cm.softCam.sepaGripperAxisX.jrWinderPos.inPos) AND "Unit1.Em7.ControlNodes".emRelations.em4.softCam.anodeMainPnP1AxisZ.avoidPos.inPos AND "Unit1.Em7.ControlNodes".emRelations.em4.softCam.anodeMainPnP2AxisZ.avoidPos.inPos,
                           int3 := "Unit1.Em7.ControlNodes".cm.softCam.sepaGripperAxisC.waitPos.inPos,
                           commands := "Unit1.Em7.HmiInterface".cmSepaGripperAxisX.commands,
                           interlockOk := "Unit1.Em7.ControlNodes".cm.interlock.sepaGripperAxisX.source.posAbsolute,
                           intOut := "Unit1.Em7.HmiInterface".intCondition.Axis_36.Jog.intOut);
   #_w1 := ((("Unit1.Em7.ControlNodes".sepaClamp."step".action2[280] OR "Unit1.Em7.ControlNodes".cm.softCam.sepaClampnCutterAxisX.winderReadyPos.inPos) AND ("Unit1.Em7.ControlNodes".sepaGripper."step".action2[280] OR "Unit1.Em7.ControlNodes".sepaGripper."step".action1[1240])) OR NOT (NOT "Unit1.Em7.ControlNodes".sepaGripper."step".action1[410] AND NOT "Unit1.Em7.ControlNodes".sepaGripper."step".action1[1511])) AND "Unit1.Em7.ControlNodes".cm.interlock.sepaGripperAxisX.source.posAbsolute[3];
   IF #_w1 THEN "Unit1.Em7.ControlNodes".cmSepaGripperAxisX.commands.selectSetPosition := 3; END_IF;
   "Unit1.Em7.ControlNodes".cm.Command.sepaGripperAxisX.posAbsolute[3] := #_w1;
END_REGION

REGION Network 114: CmSepaGripperAxisX Position Absolute Position4
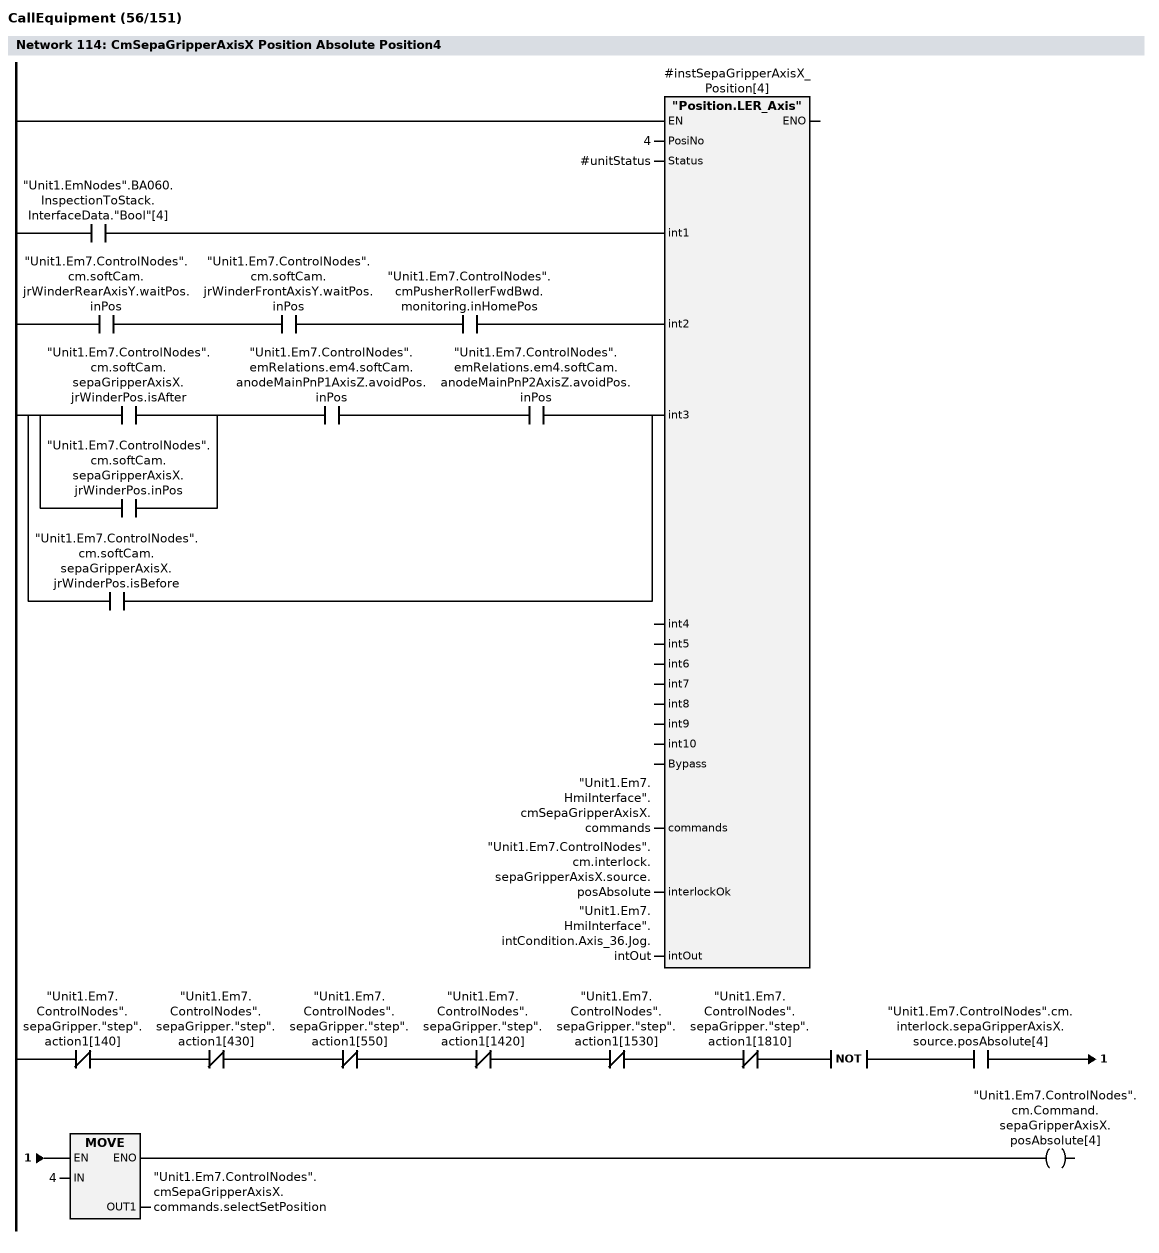
   RUNG wire#powerrail
      #instSepaGripperAxisX_Position[4](int1 := wire#w1, int2 := wire#w2, int3 := wire#w4, PosiNo := 4, Status := #unitStatus, int4 :=, int5 :=, int6 :=, int7 :=, int8 :=, int9 :=, int10 :=, Bypass :=, commands := "Unit1.Em7.HmiInterface".cmSepaGripperAxisX.commands, interlockOk := "Unit1.Em7.ControlNodes".cm.interlock.sepaGripperAxisX.source.posAbsolute, intOut := "Unit1.Em7.HmiInterface".intCondition.Axis_36.Jog.intOut)
   END_RUNG
   RUNG wire#powerrail
      Contact( "Unit1.EmNodes".BA060.InspectionToStack.InterfaceData."Bool"[4] )
   END_RUNG wire#w1
   RUNG wire#powerrail
      Contact( "Unit1.Em7.ControlNodes".cm.softCam.jrWinderRearAxisY.waitPos.inPos )
      Contact( "Unit1.Em7.ControlNodes".cm.softCam.jrWinderFrontAxisY.waitPos.inPos )
      Contact( "Unit1.Em7.ControlNodes".cmPusherRollerFwdBwd.monitoring.inHomePos )
   END_RUNG wire#w2
   RUNG wire#powerrail
      Contact( "Unit1.Em7.ControlNodes".cm.softCam.sepaGripperAxisX.jrWinderPos.isAfter )
      wire#w3
      Contact( "Unit1.Em7.ControlNodes".emRelations.em4.softCam.anodeMainPnP1AxisZ.avoidPos.inPos )
      Contact( "Unit1.Em7.ControlNodes".emRelations.em4.softCam.anodeMainPnP2AxisZ.avoidPos.inPos )
   END_RUNG wire#w4
   RUNG wire#powerrail
      Contact( "Unit1.Em7.ControlNodes".cm.softCam.sepaGripperAxisX.jrWinderPos.inPos )
   END_RUNG wire#w3
   RUNG wire#powerrail
      Contact( "Unit1.Em7.ControlNodes".cm.softCam.sepaGripperAxisX.jrWinderPos.isBefore )
   END_RUNG wire#w4
   RUNG wire#powerrail
      I_Contact( "Unit1.Em7.ControlNodes".sepaGripper."step".action1[140] )
      I_Contact( "Unit1.Em7.ControlNodes".sepaGripper."step".action1[430] )
      I_Contact( "Unit1.Em7.ControlNodes".sepaGripper."step".action1[550] )
      I_Contact( "Unit1.Em7.ControlNodes".sepaGripper."step".action1[1420] )
      I_Contact( "Unit1.Em7.ControlNodes".sepaGripper."step".action1[1530] )
      I_Contact( "Unit1.Em7.ControlNodes".sepaGripper."step".action1[1810] )
      Not()
      Contact( "Unit1.Em7.ControlNodes".cm.interlock.sepaGripperAxisX.source.posAbsolute[4] )
      Move(in := 4, out1 => "Unit1.Em7.ControlNodes".cmSepaGripperAxisX.commands.selectSetPosition)
      Coil( "Unit1.Em7.ControlNodes".cm.Command.sepaGripperAxisX.posAbsolute[4] )
   END_RUNG
   // the same network as SCL:
   #instSepaGripperAxisX_Position[4](PosiNo := 4,   // "Position.LER_Axis"
                           Status := #unitStatus,
                           int1 := "Unit1.EmNodes".BA060.InspectionToStack.InterfaceData."Bool"[4],
                           int2 := "Unit1.Em7.ControlNodes".cm.softCam.jrWinderRearAxisY.waitPos.inPos AND "Unit1.Em7.ControlNodes".cm.softCam.jrWinderFrontAxisY.waitPos.inPos AND "Unit1.Em7.ControlNodes".cmPusherRollerFwdBwd.monitoring.inHomePos,
                           int3 := (("Unit1.Em7.ControlNodes".cm.softCam.sepaGripperAxisX.jrWinderPos.isAfter OR "Unit1.Em7.ControlNodes".cm.softCam.sepaGripperAxisX.jrWinderPos.inPos) AND "Unit1.Em7.ControlNodes".emRelations.em4.softCam.anodeMainPnP1AxisZ.avoidPos.inPos AND "Unit1.Em7.ControlNodes".emRelations.em4.softCam.anodeMainPnP2AxisZ.avoidPos.inPos) OR "Unit1.Em7.ControlNodes".cm.softCam.sepaGripperAxisX.jrWinderPos.isBefore,
                           commands := "Unit1.Em7.HmiInterface".cmSepaGripperAxisX.commands,
                           interlockOk := "Unit1.Em7.ControlNodes".cm.interlock.sepaGripperAxisX.source.posAbsolute,
                           intOut := "Unit1.Em7.HmiInterface".intCondition.Axis_36.Jog.intOut);
   #_w1 := NOT (NOT "Unit1.Em7.ControlNodes".sepaGripper."step".action1[140] AND NOT "Unit1.Em7.ControlNodes".sepaGripper."step".action1[430] AND NOT "Unit1.Em7.ControlNodes".sepaGripper."step".action1[550] AND NOT "Unit1.Em7.ControlNodes".sepaGripper."step".action1[1420] AND NOT "Unit1.Em7.ControlNodes".sepaGripper."step".action1[1530] AND NOT "Unit1.Em7.ControlNodes".sepaGripper."step".action1[1810]) AND "Unit1.Em7.ControlNodes".cm.interlock.sepaGripperAxisX.source.posAbsolute[4];
   IF #_w1 THEN "Unit1.Em7.ControlNodes".cmSepaGripperAxisX.commands.selectSetPosition := 4; END_IF;
   "Unit1.Em7.ControlNodes".cm.Command.sepaGripperAxisX.posAbsolute[4] := #_w1;
END_REGION

REGION Network 115: CmSepaGripperAxisX Position Absolute Position5
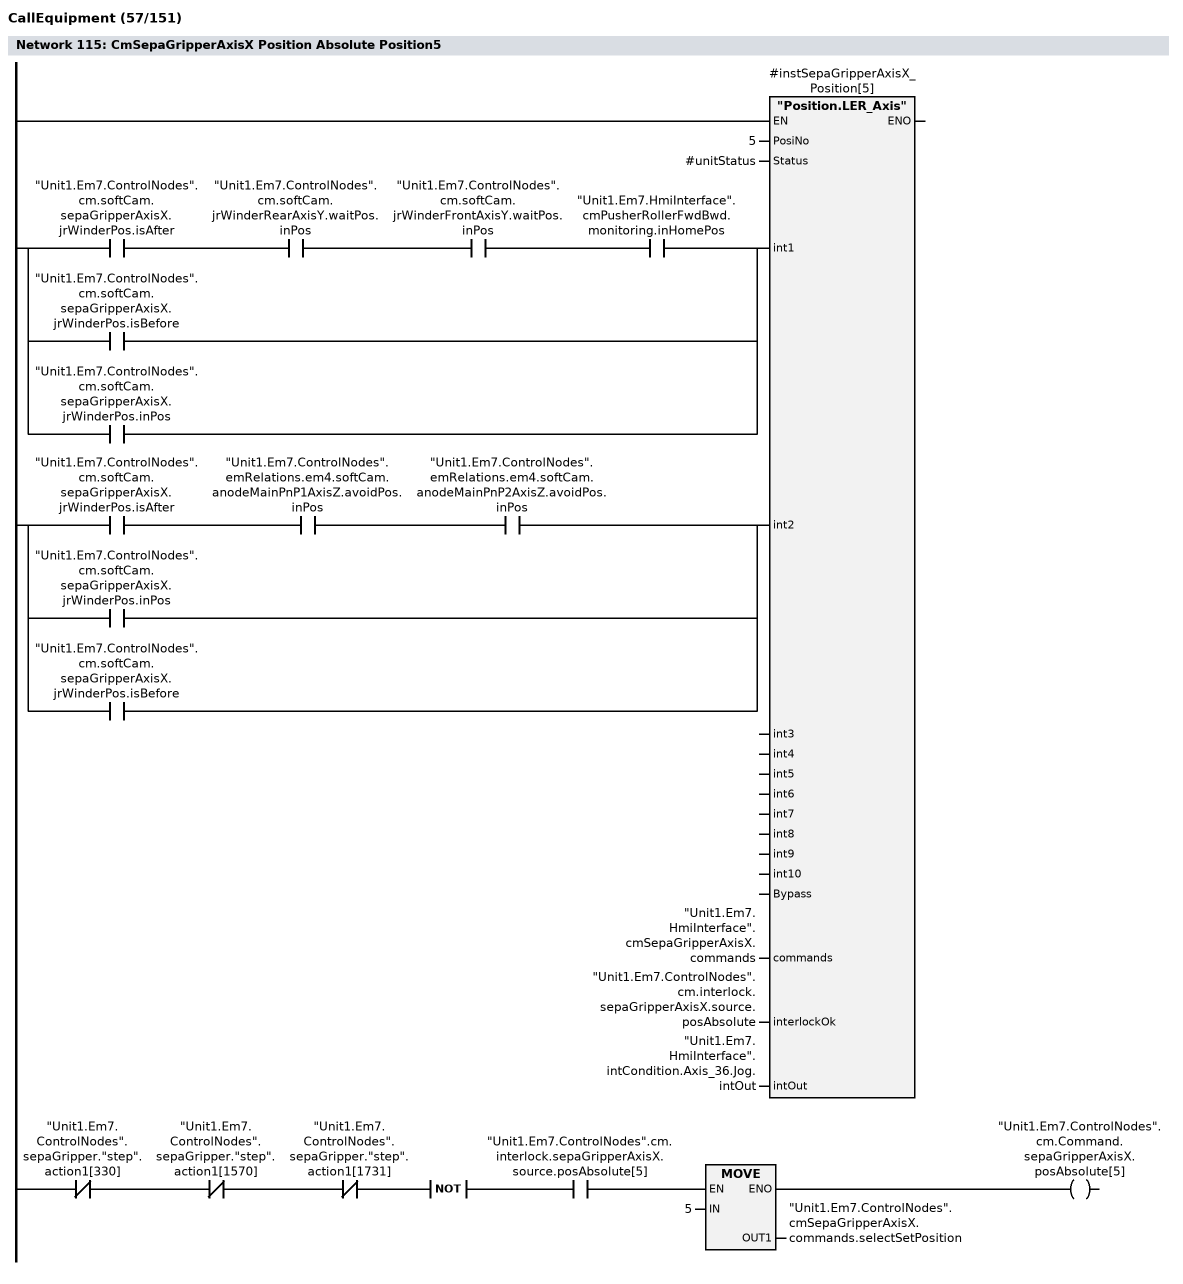
   RUNG wire#powerrail
      #instSepaGripperAxisX_Position[5](int1 := wire#w1, int2 := wire#w2, PosiNo := 5, Status := #unitStatus, int3 :=, int4 :=, int5 :=, int6 :=, int7 :=, int8 :=, int9 :=, int10 :=, Bypass :=, commands := "Unit1.Em7.HmiInterface".cmSepaGripperAxisX.commands, interlockOk := "Unit1.Em7.ControlNodes".cm.interlock.sepaGripperAxisX.source.posAbsolute, intOut := "Unit1.Em7.HmiInterface".intCondition.Axis_36.Jog.intOut)
   END_RUNG
   RUNG wire#powerrail
      Contact( "Unit1.Em7.ControlNodes".cm.softCam.sepaGripperAxisX.jrWinderPos.isAfter )
      Contact( "Unit1.Em7.ControlNodes".cm.softCam.jrWinderRearAxisY.waitPos.inPos )
      Contact( "Unit1.Em7.ControlNodes".cm.softCam.jrWinderFrontAxisY.waitPos.inPos )
      Contact( "Unit1.Em7.HmiInterface".cmPusherRollerFwdBwd.monitoring.inHomePos )
   END_RUNG wire#w1
   RUNG wire#powerrail
      Contact( "Unit1.Em7.ControlNodes".cm.softCam.sepaGripperAxisX.jrWinderPos.isBefore )
   END_RUNG wire#w1
   RUNG wire#powerrail
      Contact( "Unit1.Em7.ControlNodes".cm.softCam.sepaGripperAxisX.jrWinderPos.inPos )
   END_RUNG wire#w1
   RUNG wire#powerrail
      Contact( "Unit1.Em7.ControlNodes".cm.softCam.sepaGripperAxisX.jrWinderPos.isAfter )
      Contact( "Unit1.Em7.ControlNodes".emRelations.em4.softCam.anodeMainPnP1AxisZ.avoidPos.inPos )
      Contact( "Unit1.Em7.ControlNodes".emRelations.em4.softCam.anodeMainPnP2AxisZ.avoidPos.inPos )
   END_RUNG wire#w2
   RUNG wire#powerrail
      Contact( "Unit1.Em7.ControlNodes".cm.softCam.sepaGripperAxisX.jrWinderPos.inPos )
   END_RUNG wire#w2
   RUNG wire#powerrail
      Contact( "Unit1.Em7.ControlNodes".cm.softCam.sepaGripperAxisX.jrWinderPos.isBefore )
   END_RUNG wire#w2
   RUNG wire#powerrail
      I_Contact( "Unit1.Em7.ControlNodes".sepaGripper."step".action1[330] )
      I_Contact( "Unit1.Em7.ControlNodes".sepaGripper."step".action1[1570] )
      I_Contact( "Unit1.Em7.ControlNodes".sepaGripper."step".action1[1731] )
      Not()
      Contact( "Unit1.Em7.ControlNodes".cm.interlock.sepaGripperAxisX.source.posAbsolute[5] )
      Move(in := 5, out1 => "Unit1.Em7.ControlNodes".cmSepaGripperAxisX.commands.selectSetPosition)
      Coil( "Unit1.Em7.ControlNodes".cm.Command.sepaGripperAxisX.posAbsolute[5] )
   END_RUNG
   // the same network as SCL:
   #instSepaGripperAxisX_Position[5](PosiNo := 5,   // "Position.LER_Axis"
                           Status := #unitStatus,
                           int1 := ("Unit1.Em7.ControlNodes".cm.softCam.sepaGripperAxisX.jrWinderPos.isAfter AND "Unit1.Em7.ControlNodes".cm.softCam.jrWinderRearAxisY.waitPos.inPos AND "Unit1.Em7.ControlNodes".cm.softCam.jrWinderFrontAxisY.waitPos.inPos AND "Unit1.Em7.HmiInterface".cmPusherRollerFwdBwd.monitoring.inHomePos) OR "Unit1.Em7.ControlNodes".cm.softCam.sepaGripperAxisX.jrWinderPos.isBefore OR "Unit1.Em7.ControlNodes".cm.softCam.sepaGripperAxisX.jrWinderPos.inPos,
                           int2 := ("Unit1.Em7.ControlNodes".cm.softCam.sepaGripperAxisX.jrWinderPos.isAfter AND "Unit1.Em7.ControlNodes".emRelations.em4.softCam.anodeMainPnP1AxisZ.avoidPos.inPos AND "Unit1.Em7.ControlNodes".emRelations.em4.softCam.anodeMainPnP2AxisZ.avoidPos.inPos) OR "Unit1.Em7.ControlNodes".cm.softCam.sepaGripperAxisX.jrWinderPos.inPos OR "Unit1.Em7.ControlNodes".cm.softCam.sepaGripperAxisX.jrWinderPos.isBefore,
                           commands := "Unit1.Em7.HmiInterface".cmSepaGripperAxisX.commands,
                           interlockOk := "Unit1.Em7.ControlNodes".cm.interlock.sepaGripperAxisX.source.posAbsolute,
                           intOut := "Unit1.Em7.HmiInterface".intCondition.Axis_36.Jog.intOut);
   #_w1 := NOT (NOT "Unit1.Em7.ControlNodes".sepaGripper."step".action1[330] AND NOT "Unit1.Em7.ControlNodes".sepaGripper."step".action1[1570] AND NOT "Unit1.Em7.ControlNodes".sepaGripper."step".action1[1731]) AND "Unit1.Em7.ControlNodes".cm.interlock.sepaGripperAxisX.source.posAbsolute[5];
   IF #_w1 THEN "Unit1.Em7.ControlNodes".cmSepaGripperAxisX.commands.selectSetPosition := 5; END_IF;
   "Unit1.Em7.ControlNodes".cm.Command.sepaGripperAxisX.posAbsolute[5] := #_w1;
END_REGION

REGION Network 116: CmSepaGripperAxisX Position Absolute Position6
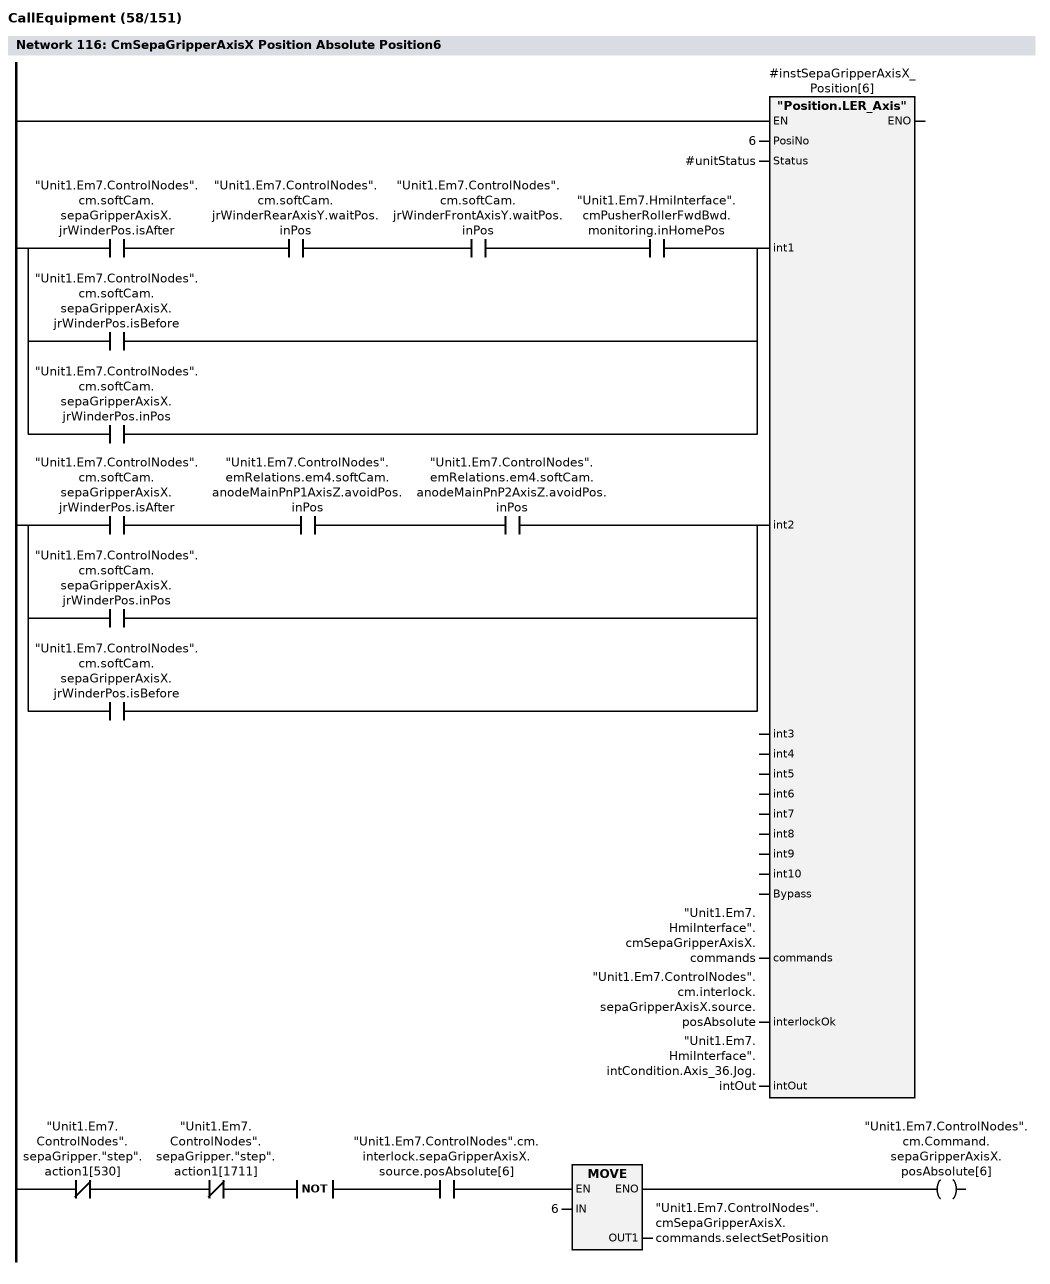
   RUNG wire#powerrail
      #instSepaGripperAxisX_Position[6](int1 := wire#w1, int2 := wire#w2, PosiNo := 6, Status := #unitStatus, int3 :=, int4 :=, int5 :=, int6 :=, int7 :=, int8 :=, int9 :=, int10 :=, Bypass :=, commands := "Unit1.Em7.HmiInterface".cmSepaGripperAxisX.commands, interlockOk := "Unit1.Em7.ControlNodes".cm.interlock.sepaGripperAxisX.source.posAbsolute, intOut := "Unit1.Em7.HmiInterface".intCondition.Axis_36.Jog.intOut)
   END_RUNG
   RUNG wire#powerrail
      Contact( "Unit1.Em7.ControlNodes".cm.softCam.sepaGripperAxisX.jrWinderPos.isAfter )
      Contact( "Unit1.Em7.ControlNodes".cm.softCam.jrWinderRearAxisY.waitPos.inPos )
      Contact( "Unit1.Em7.ControlNodes".cm.softCam.jrWinderFrontAxisY.waitPos.inPos )
      Contact( "Unit1.Em7.HmiInterface".cmPusherRollerFwdBwd.monitoring.inHomePos )
   END_RUNG wire#w1
   RUNG wire#powerrail
      Contact( "Unit1.Em7.ControlNodes".cm.softCam.sepaGripperAxisX.jrWinderPos.isBefore )
   END_RUNG wire#w1
   RUNG wire#powerrail
      Contact( "Unit1.Em7.ControlNodes".cm.softCam.sepaGripperAxisX.jrWinderPos.inPos )
   END_RUNG wire#w1
   RUNG wire#powerrail
      Contact( "Unit1.Em7.ControlNodes".cm.softCam.sepaGripperAxisX.jrWinderPos.isAfter )
      Contact( "Unit1.Em7.ControlNodes".emRelations.em4.softCam.anodeMainPnP1AxisZ.avoidPos.inPos )
      Contact( "Unit1.Em7.ControlNodes".emRelations.em4.softCam.anodeMainPnP2AxisZ.avoidPos.inPos )
   END_RUNG wire#w2
   RUNG wire#powerrail
      Contact( "Unit1.Em7.ControlNodes".cm.softCam.sepaGripperAxisX.jrWinderPos.inPos )
   END_RUNG wire#w2
   RUNG wire#powerrail
      Contact( "Unit1.Em7.ControlNodes".cm.softCam.sepaGripperAxisX.jrWinderPos.isBefore )
   END_RUNG wire#w2
   RUNG wire#powerrail
      I_Contact( "Unit1.Em7.ControlNodes".sepaGripper."step".action1[530] )
      I_Contact( "Unit1.Em7.ControlNodes".sepaGripper."step".action1[1711] )
      Not()
      Contact( "Unit1.Em7.ControlNodes".cm.interlock.sepaGripperAxisX.source.posAbsolute[6] )
      Move(in := 6, out1 => "Unit1.Em7.ControlNodes".cmSepaGripperAxisX.commands.selectSetPosition)
      Coil( "Unit1.Em7.ControlNodes".cm.Command.sepaGripperAxisX.posAbsolute[6] )
   END_RUNG
   // the same network as SCL:
   #instSepaGripperAxisX_Position[6](PosiNo := 6,   // "Position.LER_Axis"
                           Status := #unitStatus,
                           int1 := ("Unit1.Em7.ControlNodes".cm.softCam.sepaGripperAxisX.jrWinderPos.isAfter AND "Unit1.Em7.ControlNodes".cm.softCam.jrWinderRearAxisY.waitPos.inPos AND "Unit1.Em7.ControlNodes".cm.softCam.jrWinderFrontAxisY.waitPos.inPos AND "Unit1.Em7.HmiInterface".cmPusherRollerFwdBwd.monitoring.inHomePos) OR "Unit1.Em7.ControlNodes".cm.softCam.sepaGripperAxisX.jrWinderPos.isBefore OR "Unit1.Em7.ControlNodes".cm.softCam.sepaGripperAxisX.jrWinderPos.inPos,
                           int2 := ("Unit1.Em7.ControlNodes".cm.softCam.sepaGripperAxisX.jrWinderPos.isAfter AND "Unit1.Em7.ControlNodes".emRelations.em4.softCam.anodeMainPnP1AxisZ.avoidPos.inPos AND "Unit1.Em7.ControlNodes".emRelations.em4.softCam.anodeMainPnP2AxisZ.avoidPos.inPos) OR "Unit1.Em7.ControlNodes".cm.softCam.sepaGripperAxisX.jrWinderPos.inPos OR "Unit1.Em7.ControlNodes".cm.softCam.sepaGripperAxisX.jrWinderPos.isBefore,
                           commands := "Unit1.Em7.HmiInterface".cmSepaGripperAxisX.commands,
                           interlockOk := "Unit1.Em7.ControlNodes".cm.interlock.sepaGripperAxisX.source.posAbsolute,
                           intOut := "Unit1.Em7.HmiInterface".intCondition.Axis_36.Jog.intOut);
   #_w1 := NOT (NOT "Unit1.Em7.ControlNodes".sepaGripper."step".action1[530] AND NOT "Unit1.Em7.ControlNodes".sepaGripper."step".action1[1711]) AND "Unit1.Em7.ControlNodes".cm.interlock.sepaGripperAxisX.source.posAbsolute[6];
   IF #_w1 THEN "Unit1.Em7.ControlNodes".cmSepaGripperAxisX.commands.selectSetPosition := 6; END_IF;
   "Unit1.Em7.ControlNodes".cm.Command.sepaGripperAxisX.posAbsolute[6] := #_w1;
END_REGION

REGION Network 117: CmSepaGripperAxisX Position Absolute Position7
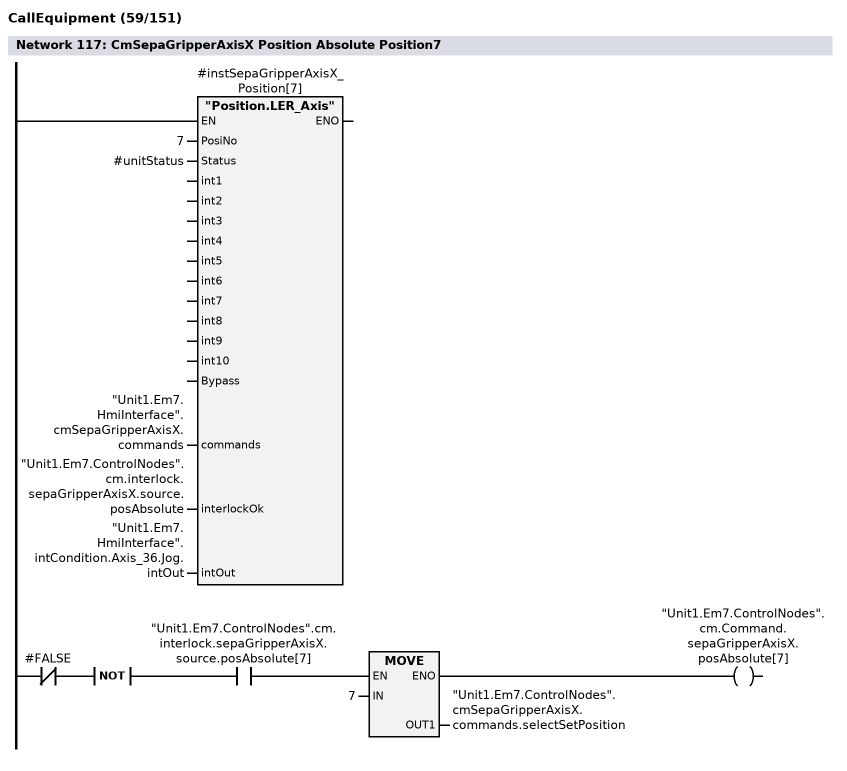
   RUNG wire#powerrail
      #instSepaGripperAxisX_Position[7](PosiNo := 7, Status := #unitStatus, int1 :=, int2 :=, int3 :=, int4 :=, int5 :=, int6 :=, int7 :=, int8 :=, int9 :=, int10 :=, Bypass :=, commands := "Unit1.Em7.HmiInterface".cmSepaGripperAxisX.commands, interlockOk := "Unit1.Em7.ControlNodes".cm.interlock.sepaGripperAxisX.source.posAbsolute, intOut := "Unit1.Em7.HmiInterface".intCondition.Axis_36.Jog.intOut)
   END_RUNG
   RUNG wire#powerrail
      I_Contact( #FALSE )
      Not()
      Contact( "Unit1.Em7.ControlNodes".cm.interlock.sepaGripperAxisX.source.posAbsolute[7] )
      Move(in := 7, out1 => "Unit1.Em7.ControlNodes".cmSepaGripperAxisX.commands.selectSetPosition)
      Coil( "Unit1.Em7.ControlNodes".cm.Command.sepaGripperAxisX.posAbsolute[7] )
   END_RUNG
   // the same network as SCL:
   #instSepaGripperAxisX_Position[7](PosiNo := 7,   // "Position.LER_Axis"
                           Status := #unitStatus,
                           commands := "Unit1.Em7.HmiInterface".cmSepaGripperAxisX.commands,
                           interlockOk := "Unit1.Em7.ControlNodes".cm.interlock.sepaGripperAxisX.source.posAbsolute,
                           intOut := "Unit1.Em7.HmiInterface".intCondition.Axis_36.Jog.intOut);
   #_w1 := NOT (NOT #FALSE) AND "Unit1.Em7.ControlNodes".cm.interlock.sepaGripperAxisX.source.posAbsolute[7];
   IF #_w1 THEN "Unit1.Em7.ControlNodes".cmSepaGripperAxisX.commands.selectSetPosition := 7; END_IF;
   "Unit1.Em7.ControlNodes".cm.Command.sepaGripperAxisX.posAbsolute[7] := #_w1;
END_REGION

REGION Network 118: CmSepaGripperAxisX Position Absolute Position8
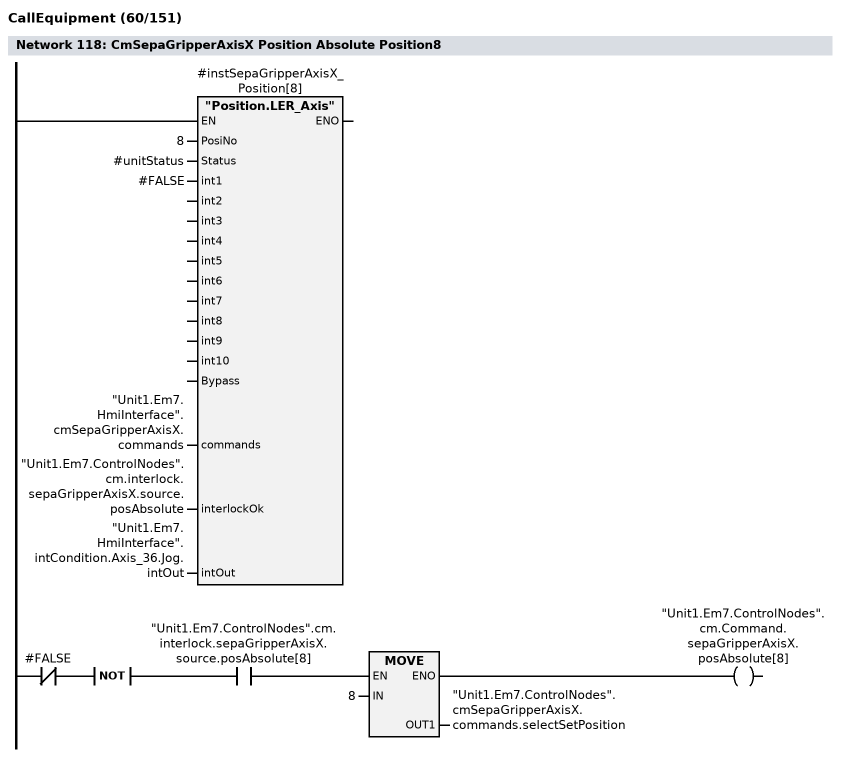
   RUNG wire#powerrail
      #instSepaGripperAxisX_Position[8](PosiNo := 8, Status := #unitStatus, int1 := #FALSE, int2 :=, int3 :=, int4 :=, int5 :=, int6 :=, int7 :=, int8 :=, int9 :=, int10 :=, Bypass :=, commands := "Unit1.Em7.HmiInterface".cmSepaGripperAxisX.commands, interlockOk := "Unit1.Em7.ControlNodes".cm.interlock.sepaGripperAxisX.source.posAbsolute, intOut := "Unit1.Em7.HmiInterface".intCondition.Axis_36.Jog.intOut)
   END_RUNG
   RUNG wire#powerrail
      I_Contact( #FALSE )
      Not()
      Contact( "Unit1.Em7.ControlNodes".cm.interlock.sepaGripperAxisX.source.posAbsolute[8] )
      Move(in := 8, out1 => "Unit1.Em7.ControlNodes".cmSepaGripperAxisX.commands.selectSetPosition)
      Coil( "Unit1.Em7.ControlNodes".cm.Command.sepaGripperAxisX.posAbsolute[8] )
   END_RUNG
   // the same network as SCL:
   #instSepaGripperAxisX_Position[8](PosiNo := 8,   // "Position.LER_Axis"
                           Status := #unitStatus,
                           int1 := #FALSE,
                           commands := "Unit1.Em7.HmiInterface".cmSepaGripperAxisX.commands,
                           interlockOk := "Unit1.Em7.ControlNodes".cm.interlock.sepaGripperAxisX.source.posAbsolute,
                           intOut := "Unit1.Em7.HmiInterface".intCondition.Axis_36.Jog.intOut);
   #_w1 := NOT (NOT #FALSE) AND "Unit1.Em7.ControlNodes".cm.interlock.sepaGripperAxisX.source.posAbsolute[8];
   IF #_w1 THEN "Unit1.Em7.ControlNodes".cmSepaGripperAxisX.commands.selectSetPosition := 8; END_IF;
   "Unit1.Em7.ControlNodes".cm.Command.sepaGripperAxisX.posAbsolute[8] := #_w1;
END_REGION

REGION Network 119: CmSepaGripperAxisX Position Absolute Position9
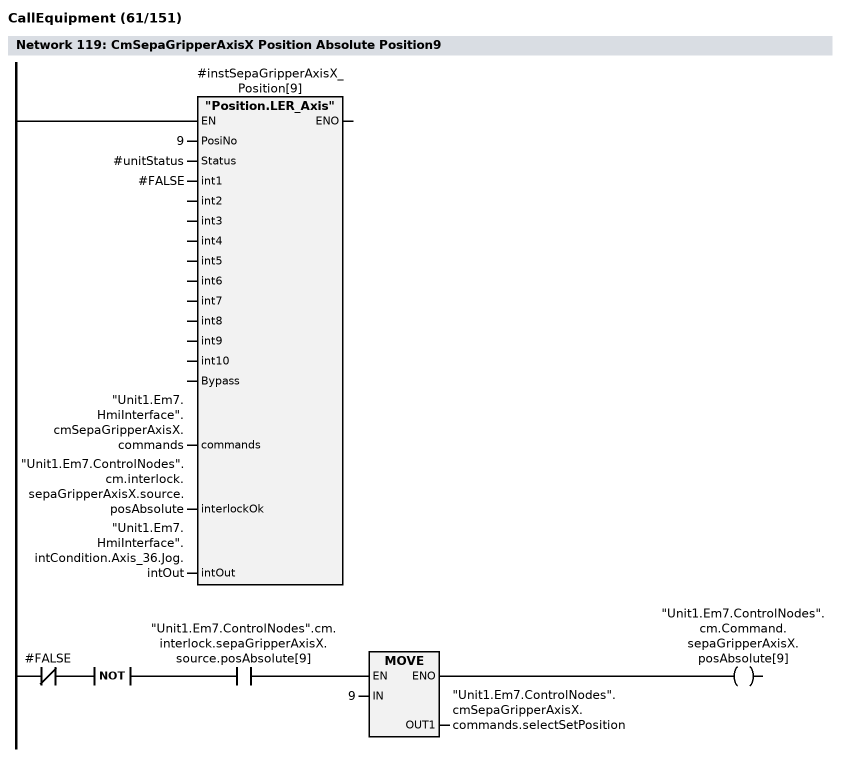
   RUNG wire#powerrail
      #instSepaGripperAxisX_Position[9](PosiNo := 9, Status := #unitStatus, int1 := #FALSE, int2 :=, int3 :=, int4 :=, int5 :=, int6 :=, int7 :=, int8 :=, int9 :=, int10 :=, Bypass :=, commands := "Unit1.Em7.HmiInterface".cmSepaGripperAxisX.commands, interlockOk := "Unit1.Em7.ControlNodes".cm.interlock.sepaGripperAxisX.source.posAbsolute, intOut := "Unit1.Em7.HmiInterface".intCondition.Axis_36.Jog.intOut)
   END_RUNG
   RUNG wire#powerrail
      I_Contact( #FALSE )
      Not()
      Contact( "Unit1.Em7.ControlNodes".cm.interlock.sepaGripperAxisX.source.posAbsolute[9] )
      Move(in := 9, out1 => "Unit1.Em7.ControlNodes".cmSepaGripperAxisX.commands.selectSetPosition)
      Coil( "Unit1.Em7.ControlNodes".cm.Command.sepaGripperAxisX.posAbsolute[9] )
   END_RUNG
   // the same network as SCL:
   #instSepaGripperAxisX_Position[9](PosiNo := 9,   // "Position.LER_Axis"
                           Status := #unitStatus,
                           int1 := #FALSE,
                           commands := "Unit1.Em7.HmiInterface".cmSepaGripperAxisX.commands,
                           interlockOk := "Unit1.Em7.ControlNodes".cm.interlock.sepaGripperAxisX.source.posAbsolute,
                           intOut := "Unit1.Em7.HmiInterface".intCondition.Axis_36.Jog.intOut);
   #_w1 := NOT (NOT #FALSE) AND "Unit1.Em7.ControlNodes".cm.interlock.sepaGripperAxisX.source.posAbsolute[9];
   IF #_w1 THEN "Unit1.Em7.ControlNodes".cmSepaGripperAxisX.commands.selectSetPosition := 9; END_IF;
   "Unit1.Em7.ControlNodes".cm.Command.sepaGripperAxisX.posAbsolute[9] := #_w1;
END_REGION

REGION Network 120: CmSepaGripperAxisX Position Absolute Position10
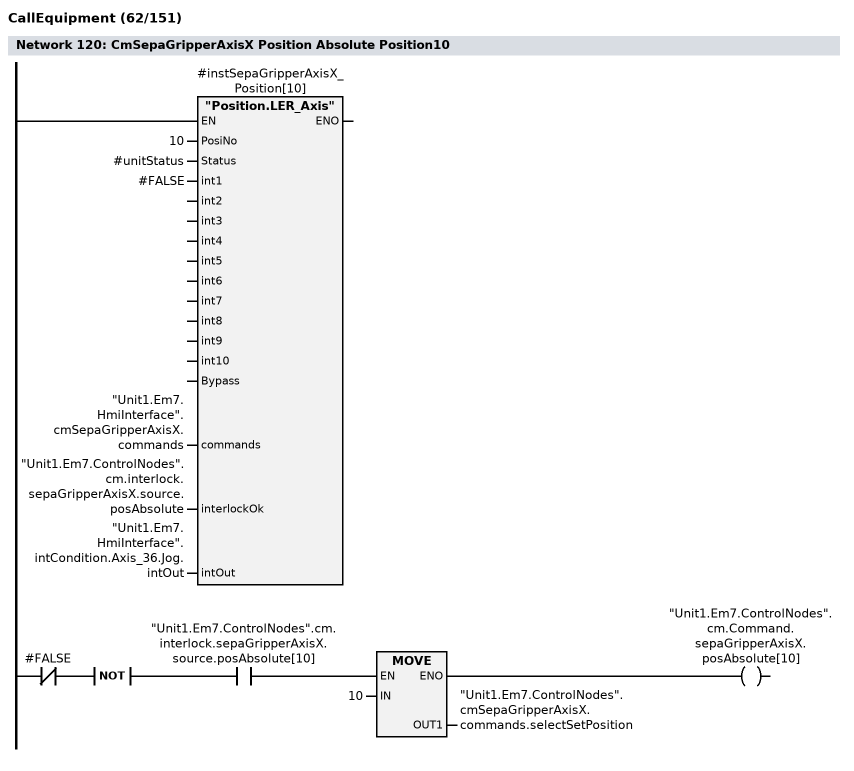
   RUNG wire#powerrail
      #instSepaGripperAxisX_Position[10](PosiNo := 10, Status := #unitStatus, int1 := #FALSE, int2 :=, int3 :=, int4 :=, int5 :=, int6 :=, int7 :=, int8 :=, int9 :=, int10 :=, Bypass :=, commands := "Unit1.Em7.HmiInterface".cmSepaGripperAxisX.commands, interlockOk := "Unit1.Em7.ControlNodes".cm.interlock.sepaGripperAxisX.source.posAbsolute, intOut := "Unit1.Em7.HmiInterface".intCondition.Axis_36.Jog.intOut)
   END_RUNG
   RUNG wire#powerrail
      I_Contact( #FALSE )
      Not()
      Contact( "Unit1.Em7.ControlNodes".cm.interlock.sepaGripperAxisX.source.posAbsolute[10] )
      Move(in := 10, out1 => "Unit1.Em7.ControlNodes".cmSepaGripperAxisX.commands.selectSetPosition)
      Coil( "Unit1.Em7.ControlNodes".cm.Command.sepaGripperAxisX.posAbsolute[10] )
   END_RUNG
   // the same network as SCL:
   #instSepaGripperAxisX_Position[10](PosiNo := 10,   // "Position.LER_Axis"
                           Status := #unitStatus,
                           int1 := #FALSE,
                           commands := "Unit1.Em7.HmiInterface".cmSepaGripperAxisX.commands,
                           interlockOk := "Unit1.Em7.ControlNodes".cm.interlock.sepaGripperAxisX.source.posAbsolute,
                           intOut := "Unit1.Em7.HmiInterface".intCondition.Axis_36.Jog.intOut);
   #_w1 := NOT (NOT #FALSE) AND "Unit1.Em7.ControlNodes".cm.interlock.sepaGripperAxisX.source.posAbsolute[10];
   IF #_w1 THEN "Unit1.Em7.ControlNodes".cmSepaGripperAxisX.commands.selectSetPosition := 10; END_IF;
   "Unit1.Em7.ControlNodes".cm.Command.sepaGripperAxisX.posAbsolute[10] := #_w1;
END_REGION

REGION Network 121: CmSepaGripperAxisX Position Absolute Position11
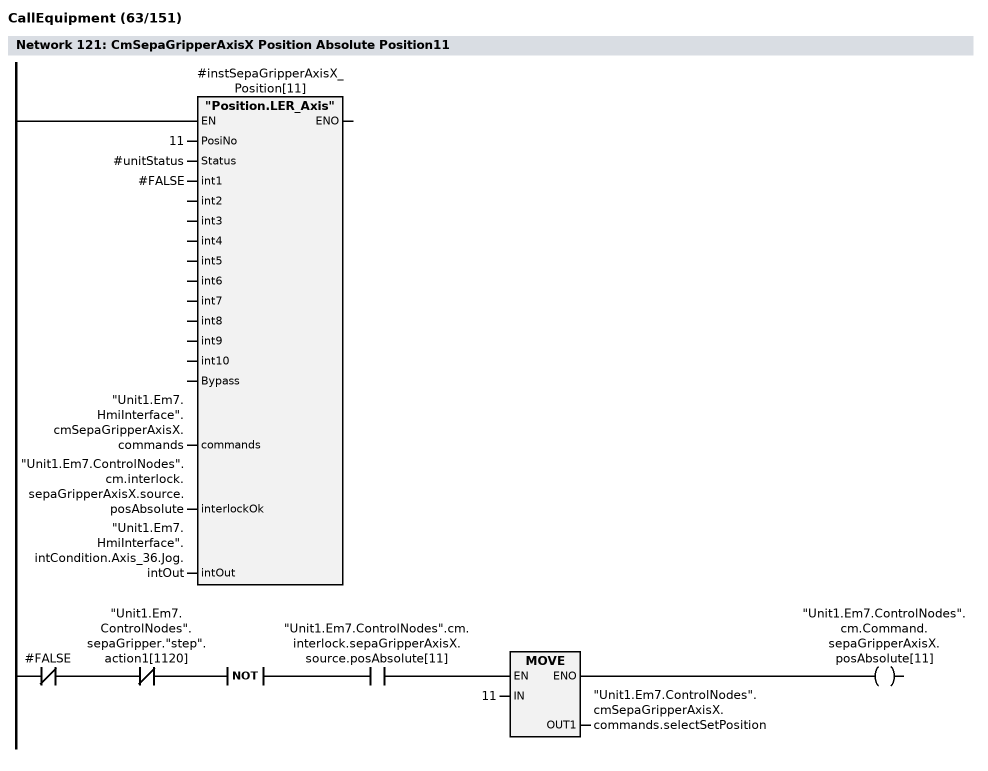
   RUNG wire#powerrail
      #instSepaGripperAxisX_Position[11](PosiNo := 11, Status := #unitStatus, int1 := #FALSE, int2 :=, int3 :=, int4 :=, int5 :=, int6 :=, int7 :=, int8 :=, int9 :=, int10 :=, Bypass :=, commands := "Unit1.Em7.HmiInterface".cmSepaGripperAxisX.commands, interlockOk := "Unit1.Em7.ControlNodes".cm.interlock.sepaGripperAxisX.source.posAbsolute, intOut := "Unit1.Em7.HmiInterface".intCondition.Axis_36.Jog.intOut)
   END_RUNG
   RUNG wire#powerrail
      I_Contact( #FALSE )
      I_Contact( "Unit1.Em7.ControlNodes".sepaGripper."step".action1[1120] )
      Not()
      Contact( "Unit1.Em7.ControlNodes".cm.interlock.sepaGripperAxisX.source.posAbsolute[11] )
      Move(in := 11, out1 => "Unit1.Em7.ControlNodes".cmSepaGripperAxisX.commands.selectSetPosition)
      Coil( "Unit1.Em7.ControlNodes".cm.Command.sepaGripperAxisX.posAbsolute[11] )
   END_RUNG
   // the same network as SCL:
   #instSepaGripperAxisX_Position[11](PosiNo := 11,   // "Position.LER_Axis"
                           Status := #unitStatus,
                           int1 := #FALSE,
                           commands := "Unit1.Em7.HmiInterface".cmSepaGripperAxisX.commands,
                           interlockOk := "Unit1.Em7.ControlNodes".cm.interlock.sepaGripperAxisX.source.posAbsolute,
                           intOut := "Unit1.Em7.HmiInterface".intCondition.Axis_36.Jog.intOut);
   #_w1 := NOT (NOT #FALSE AND NOT "Unit1.Em7.ControlNodes".sepaGripper."step".action1[1120]) AND "Unit1.Em7.ControlNodes".cm.interlock.sepaGripperAxisX.source.posAbsolute[11];
   IF #_w1 THEN "Unit1.Em7.ControlNodes".cmSepaGripperAxisX.commands.selectSetPosition := 11; END_IF;
   "Unit1.Em7.ControlNodes".cm.Command.sepaGripperAxisX.posAbsolute[11] := #_w1;
END_REGION

REGION Network 122: CmSepaGripperAxisX Position Absolute Position12
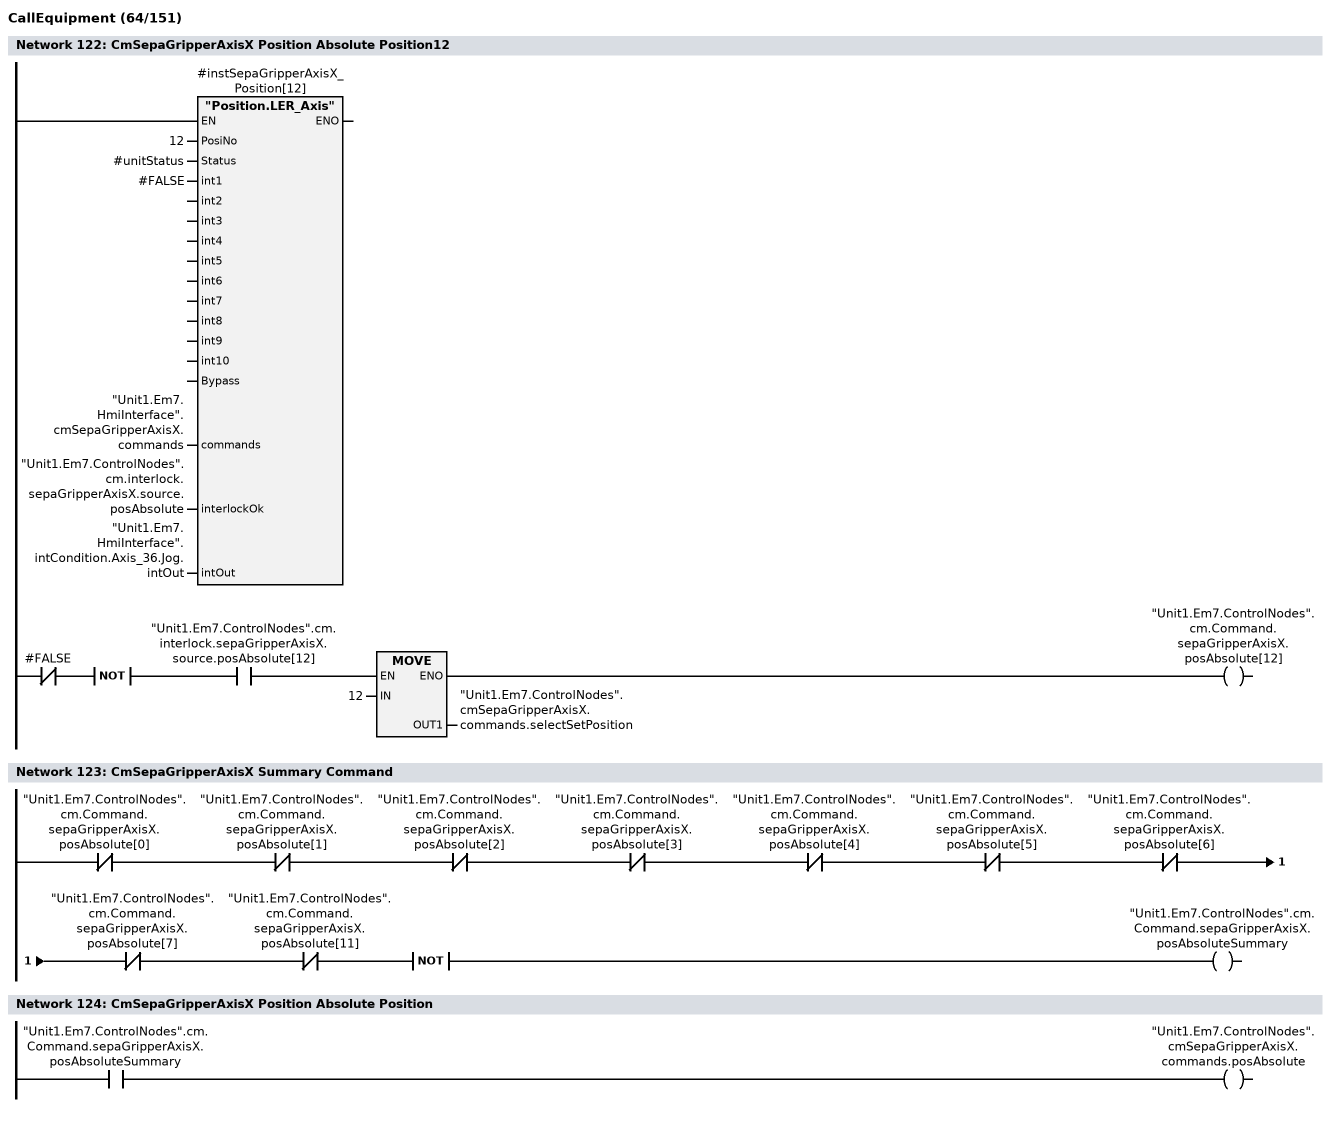
   RUNG wire#powerrail
      #instSepaGripperAxisX_Position[12](PosiNo := 12, Status := #unitStatus, int1 := #FALSE, int2 :=, int3 :=, int4 :=, int5 :=, int6 :=, int7 :=, int8 :=, int9 :=, int10 :=, Bypass :=, commands := "Unit1.Em7.HmiInterface".cmSepaGripperAxisX.commands, interlockOk := "Unit1.Em7.ControlNodes".cm.interlock.sepaGripperAxisX.source.posAbsolute, intOut := "Unit1.Em7.HmiInterface".intCondition.Axis_36.Jog.intOut)
   END_RUNG
   RUNG wire#powerrail
      I_Contact( #FALSE )
      Not()
      Contact( "Unit1.Em7.ControlNodes".cm.interlock.sepaGripperAxisX.source.posAbsolute[12] )
      Move(in := 12, out1 => "Unit1.Em7.ControlNodes".cmSepaGripperAxisX.commands.selectSetPosition)
      Coil( "Unit1.Em7.ControlNodes".cm.Command.sepaGripperAxisX.posAbsolute[12] )
   END_RUNG
   // the same network as SCL:
   #instSepaGripperAxisX_Position[12](PosiNo := 12,   // "Position.LER_Axis"
                           Status := #unitStatus,
                           int1 := #FALSE,
                           commands := "Unit1.Em7.HmiInterface".cmSepaGripperAxisX.commands,
                           interlockOk := "Unit1.Em7.ControlNodes".cm.interlock.sepaGripperAxisX.source.posAbsolute,
                           intOut := "Unit1.Em7.HmiInterface".intCondition.Axis_36.Jog.intOut);
   #_w1 := NOT (NOT #FALSE) AND "Unit1.Em7.ControlNodes".cm.interlock.sepaGripperAxisX.source.posAbsolute[12];
   IF #_w1 THEN "Unit1.Em7.ControlNodes".cmSepaGripperAxisX.commands.selectSetPosition := 12; END_IF;
   "Unit1.Em7.ControlNodes".cm.Command.sepaGripperAxisX.posAbsolute[12] := #_w1;
END_REGION

REGION Network 123: CmSepaGripperAxisX Summary Command
   RUNG wire#powerrail
      I_Contact( "Unit1.Em7.ControlNodes".cm.Command.sepaGripperAxisX.posAbsolute[0] )
      I_Contact( "Unit1.Em7.ControlNodes".cm.Command.sepaGripperAxisX.posAbsolute[1] )
      I_Contact( "Unit1.Em7.ControlNodes".cm.Command.sepaGripperAxisX.posAbsolute[2] )
      I_Contact( "Unit1.Em7.ControlNodes".cm.Command.sepaGripperAxisX.posAbsolute[3] )
      I_Contact( "Unit1.Em7.ControlNodes".cm.Command.sepaGripperAxisX.posAbsolute[4] )
      I_Contact( "Unit1.Em7.ControlNodes".cm.Command.sepaGripperAxisX.posAbsolute[5] )
      I_Contact( "Unit1.Em7.ControlNodes".cm.Command.sepaGripperAxisX.posAbsolute[6] )
      I_Contact( "Unit1.Em7.ControlNodes".cm.Command.sepaGripperAxisX.posAbsolute[7] )
      I_Contact( "Unit1.Em7.ControlNodes".cm.Command.sepaGripperAxisX.posAbsolute[11] )
      Not()
      Coil( "Unit1.Em7.ControlNodes".cm.Command.sepaGripperAxisX.posAbsoluteSummary )
   END_RUNG
   // the same network as SCL:
   "Unit1.Em7.ControlNodes".cm.Command.sepaGripperAxisX.posAbsoluteSummary := NOT (NOT "Unit1.Em7.ControlNodes".cm.Command.sepaGripperAxisX.posAbsolute[0] AND NOT "Unit1.Em7.ControlNodes".cm.Command.sepaGripperAxisX.posAbsolute[1] AND NOT "Unit1.Em7.ControlNodes".cm.Command.sepaGripperAxisX.posAbsolute[2] AND NOT "Unit1.Em7.ControlNodes".cm.Command.sepaGripperAxisX.posAbsolute[3] AND NOT "Unit1.Em7.ControlNodes".cm.Command.sepaGripperAxisX.posAbsolute[4] AND NOT "Unit1.Em7.ControlNodes".cm.Command.sepaGripperAxisX.posAbsolute[5] AND NOT "Unit1.Em7.ControlNodes".cm.Command.sepaGripperAxisX.posAbsolute[6] AND NOT "Unit1.Em7.ControlNodes".cm.Command.sepaGripperAxisX.posAbsolute[7] AND NOT "Unit1.Em7.ControlNodes".cm.Command.sepaGripperAxisX.posAbsolute[11]);
END_REGION

REGION Network 124: CmSepaGripperAxisX Position Absolute Position
   RUNG wire#powerrail
      Contact( "Unit1.Em7.ControlNodes".cm.Command.sepaGripperAxisX.posAbsoluteSummary )
      Coil( "Unit1.Em7.ControlNodes".cmSepaGripperAxisX.commands.posAbsolute )
   END_RUNG
   // the same network as SCL:
   "Unit1.Em7.ControlNodes".cmSepaGripperAxisX.commands.posAbsolute := "Unit1.Em7.ControlNodes".cm.Command.sepaGripperAxisX.posAbsoluteSummary;
END_REGION

REGION Network 125: CmSepaGripperAxisX Interlock Summary
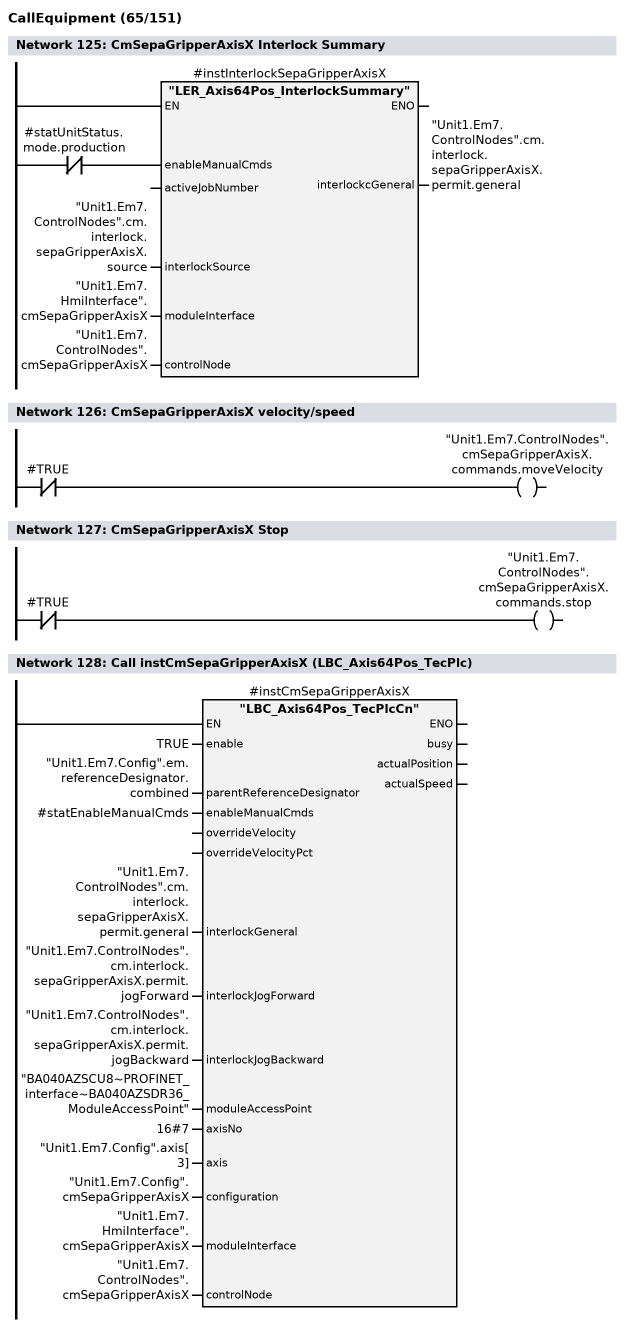
   RUNG wire#powerrail
      #instInterlockSepaGripperAxisX(enableManualCmds := wire#w1, activeJobNumber :=, interlockSource := "Unit1.Em7.ControlNodes".cm.interlock.sepaGripperAxisX.source, moduleInterface := "Unit1.Em7.HmiInterface".cmSepaGripperAxisX, controlNode := "Unit1.Em7.ControlNodes".cmSepaGripperAxisX, interlockcGeneral => "Unit1.Em7.ControlNodes".cm.interlock.sepaGripperAxisX.permit.general)
   END_RUNG
   RUNG wire#powerrail
      I_Contact( #statUnitStatus.mode.production )
   END_RUNG wire#w1
   // the same network as SCL:
   #instInterlockSepaGripperAxisX(enableManualCmds := NOT #statUnitStatus.mode.production,   // "LER_Axis64Pos_InterlockSummary"
                           interlockSource := "Unit1.Em7.ControlNodes".cm.interlock.sepaGripperAxisX.source,
                           moduleInterface := "Unit1.Em7.HmiInterface".cmSepaGripperAxisX,
                           controlNode := "Unit1.Em7.ControlNodes".cmSepaGripperAxisX,
                           interlockcGeneral => "Unit1.Em7.ControlNodes".cm.interlock.sepaGripperAxisX.permit.general);
END_REGION

REGION Network 126: CmSepaGripperAxisX velocity/speed
   RUNG wire#powerrail
      I_Contact( #TRUE )
      Coil( "Unit1.Em7.ControlNodes".cmSepaGripperAxisX.commands.moveVelocity )
   END_RUNG
   // the same network as SCL:
   "Unit1.Em7.ControlNodes".cmSepaGripperAxisX.commands.moveVelocity := NOT #TRUE;
END_REGION

REGION Network 127: CmSepaGripperAxisX Stop
   RUNG wire#powerrail
      I_Contact( #TRUE )
      Coil( "Unit1.Em7.ControlNodes".cmSepaGripperAxisX.commands.stop )
   END_RUNG
   // the same network as SCL:
   "Unit1.Em7.ControlNodes".cmSepaGripperAxisX.commands.stop := NOT #TRUE;
END_REGION

REGION Network 128: Call instCmSepaGripperAxisX (LBC_Axis64Pos_TecPlc)
   RUNG wire#powerrail
      #instCmSepaGripperAxisX(enable := TRUE, parentReferenceDesignator := "Unit1.Em7.Config".em.referenceDesignator.combined, enableManualCmds := #statEnableManualCmds, overrideVelocity :=, overrideVelocityPct :=, interlockGeneral := "Unit1.Em7.ControlNodes".cm.interlock.sepaGripperAxisX.permit.general, interlockJogForward := "Unit1.Em7.ControlNodes".cm.interlock.sepaGripperAxisX.permit.jogForward, interlockJogBackward := "Unit1.Em7.ControlNodes".cm.interlock.sepaGripperAxisX.permit.jogBackward, moduleAccessPoint := "BA040AZSCU8~PROFINET_interface~BA040AZSDR36_ModuleAccessPoint", axisNo := 16#7, axis := "Unit1.Em7.Config".axis[3], configuration := "Unit1.Em7.Config".cmSepaGripperAxisX, moduleInterface := "Unit1.Em7.HmiInterface".cmSepaGripperAxisX, controlNode := "Unit1.Em7.ControlNodes".cmSepaGripperAxisX, busy =>, actualPosition =>, actualSpeed =>)
   END_RUNG
   // the same network as SCL:
   #instCmSepaGripperAxisX(enable := TRUE,   // "LBC_Axis64Pos_TecPlcCn"
                           parentReferenceDesignator := "Unit1.Em7.Config".em.referenceDesignator.combined,
                           enableManualCmds := #statEnableManualCmds,
                           interlockGeneral := "Unit1.Em7.ControlNodes".cm.interlock.sepaGripperAxisX.permit.general,
                           interlockJogForward := "Unit1.Em7.ControlNodes".cm.interlock.sepaGripperAxisX.permit.jogForward,
                           interlockJogBackward := "Unit1.Em7.ControlNodes".cm.interlock.sepaGripperAxisX.permit.jogBackward,
                           moduleAccessPoint := "BA040AZSCU8~PROFINET_interface~BA040AZSDR36_ModuleAccessPoint",
                           axisNo := 16#7,
                           axis := "Unit1.Em7.Config".axis[3],
                           configuration := "Unit1.Em7.Config".cmSepaGripperAxisX,
                           moduleInterface := "Unit1.Em7.HmiInterface".cmSepaGripperAxisX,
                           controlNode := "Unit1.Em7.ControlNodes".cmSepaGripperAxisX);
END_REGION

REGION Network 129: CmSepaGripperAxisX SoftCam
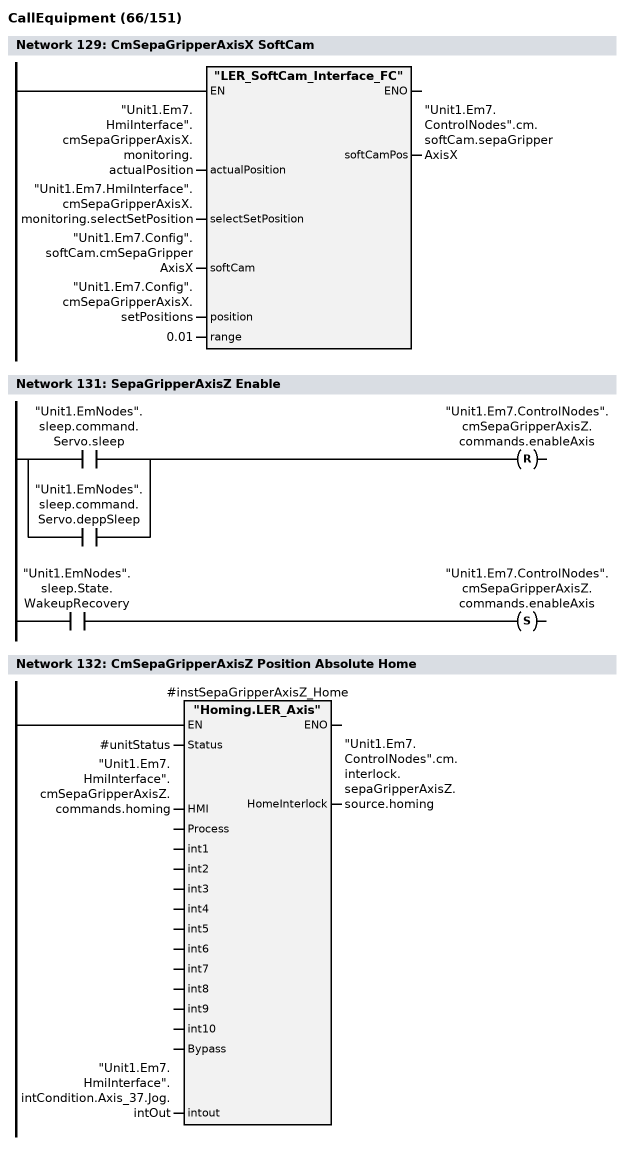
   RUNG wire#powerrail
      "LER_SoftCam_Interface_FC"(actualPosition := "Unit1.Em7.HmiInterface".cmSepaGripperAxisX.monitoring.actualPosition, selectSetPosition := "Unit1.Em7.HmiInterface".cmSepaGripperAxisX.monitoring.selectSetPosition, softCam := "Unit1.Em7.Config".softCam.cmSepaGripperAxisX, position := "Unit1.Em7.Config".cmSepaGripperAxisX.setPositions, range := 0.01, softCamPos => "Unit1.Em7.ControlNodes".cm.softCam.sepaGripperAxisX)
   END_RUNG
   // the same network as SCL:
   "LER_SoftCam_Interface_FC"(actualPosition := "Unit1.Em7.HmiInterface".cmSepaGripperAxisX.monitoring.actualPosition,
                           selectSetPosition := "Unit1.Em7.HmiInterface".cmSepaGripperAxisX.monitoring.selectSetPosition,
                           softCam := "Unit1.Em7.Config".softCam.cmSepaGripperAxisX,
                           position := "Unit1.Em7.Config".cmSepaGripperAxisX.setPositions,
                           range := 0.01,
                           softCamPos => "Unit1.Em7.ControlNodes".cm.softCam.sepaGripperAxisX);
END_REGION

REGION Network 131: SepaGripperAxisZ Enable
   RUNG wire#powerrail
      Contact( "Unit1.EmNodes".sleep.command.Servo.sleep )
      wire#w1
      R_Coil( "Unit1.Em7.ControlNodes".cmSepaGripperAxisZ.commands.enableAxis )
   END_RUNG
   RUNG wire#powerrail
      Contact( "Unit1.EmNodes".sleep.command.Servo.deppSleep )
   END_RUNG wire#w1
   RUNG wire#powerrail
      Contact( "Unit1.EmNodes".sleep.State.WakeupRecovery )
      S_Coil( "Unit1.Em7.ControlNodes".cmSepaGripperAxisZ.commands.enableAxis )
   END_RUNG
   // the same network as SCL:
   IF "Unit1.EmNodes".sleep.command.Servo.sleep OR "Unit1.EmNodes".sleep.command.Servo.deppSleep THEN
       "Unit1.Em7.ControlNodes".cmSepaGripperAxisZ.commands.enableAxis := FALSE;
   END_IF;
   IF "Unit1.EmNodes".sleep.State.WakeupRecovery THEN
       "Unit1.Em7.ControlNodes".cmSepaGripperAxisZ.commands.enableAxis := TRUE;
   END_IF;
END_REGION

REGION Network 132: CmSepaGripperAxisZ Position Absolute Home
   RUNG wire#powerrail
      #instSepaGripperAxisZ_Home(Status := #unitStatus, HMI := "Unit1.Em7.HmiInterface".cmSepaGripperAxisZ.commands.homing, Process :=, int1 :=, int2 :=, int3 :=, int4 :=, int5 :=, int6 :=, int7 :=, int8 :=, int9 :=, int10 :=, Bypass :=, intout := "Unit1.Em7.HmiInterface".intCondition.Axis_37.Jog.intOut, HomeInterlock => "Unit1.Em7.ControlNodes".cm.interlock.sepaGripperAxisZ.source.homing)
   END_RUNG
   // the same network as SCL:
   #instSepaGripperAxisZ_Home(Status := #unitStatus,   // "Homing.LER_Axis"
                           HMI := "Unit1.Em7.HmiInterface".cmSepaGripperAxisZ.commands.homing,
                           intout := "Unit1.Em7.HmiInterface".intCondition.Axis_37.Jog.intOut,
                           HomeInterlock => "Unit1.Em7.ControlNodes".cm.interlock.sepaGripperAxisZ.source.homing);
END_REGION

REGION Network 133: CmSepaGripperAxisZ Position Absolute Jog
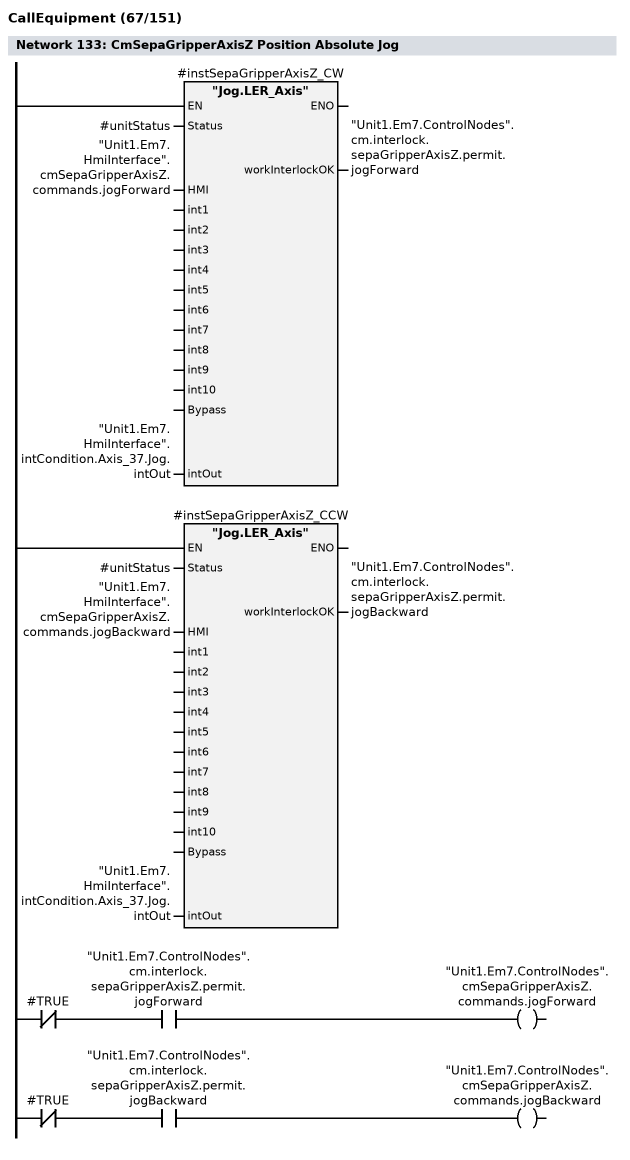
   RUNG wire#powerrail
      #instSepaGripperAxisZ_CW(Status := #unitStatus, HMI := "Unit1.Em7.HmiInterface".cmSepaGripperAxisZ.commands.jogForward, int1 :=, int2 :=, int3 :=, int4 :=, int5 :=, int6 :=, int7 :=, int8 :=, int9 :=, int10 :=, Bypass :=, intOut := "Unit1.Em7.HmiInterface".intCondition.Axis_37.Jog.intOut, workInterlockOK => "Unit1.Em7.ControlNodes".cm.interlock.sepaGripperAxisZ.permit.jogForward)
   END_RUNG
   RUNG wire#powerrail
      #instSepaGripperAxisZ_CCW(Status := #unitStatus, HMI := "Unit1.Em7.HmiInterface".cmSepaGripperAxisZ.commands.jogBackward, int1 :=, int2 :=, int3 :=, int4 :=, int5 :=, int6 :=, int7 :=, int8 :=, int9 :=, int10 :=, Bypass :=, intOut := "Unit1.Em7.HmiInterface".intCondition.Axis_37.Jog.intOut, workInterlockOK => "Unit1.Em7.ControlNodes".cm.interlock.sepaGripperAxisZ.permit.jogBackward)
   END_RUNG
   RUNG wire#powerrail
      I_Contact( #TRUE )
      Contact( "Unit1.Em7.ControlNodes".cm.interlock.sepaGripperAxisZ.permit.jogForward )
      Coil( "Unit1.Em7.ControlNodes".cmSepaGripperAxisZ.commands.jogForward )
   END_RUNG
   RUNG wire#powerrail
      I_Contact( #TRUE )
      Contact( "Unit1.Em7.ControlNodes".cm.interlock.sepaGripperAxisZ.permit.jogBackward )
      Coil( "Unit1.Em7.ControlNodes".cmSepaGripperAxisZ.commands.jogBackward )
   END_RUNG
   // the same network as SCL:
   #instSepaGripperAxisZ_CW(Status := #unitStatus,   // "Jog.LER_Axis"
                           HMI := "Unit1.Em7.HmiInterface".cmSepaGripperAxisZ.commands.jogForward,
                           intOut := "Unit1.Em7.HmiInterface".intCondition.Axis_37.Jog.intOut,
                           workInterlockOK => "Unit1.Em7.ControlNodes".cm.interlock.sepaGripperAxisZ.permit.jogForward);
   #instSepaGripperAxisZ_CCW(Status := #unitStatus,   // "Jog.LER_Axis"
                           HMI := "Unit1.Em7.HmiInterface".cmSepaGripperAxisZ.commands.jogBackward,
                           intOut := "Unit1.Em7.HmiInterface".intCondition.Axis_37.Jog.intOut,
                           workInterlockOK => "Unit1.Em7.ControlNodes".cm.interlock.sepaGripperAxisZ.permit.jogBackward);
   "Unit1.Em7.ControlNodes".cmSepaGripperAxisZ.commands.jogForward := NOT #TRUE AND "Unit1.Em7.ControlNodes".cm.interlock.sepaGripperAxisZ.permit.jogForward;
   "Unit1.Em7.ControlNodes".cmSepaGripperAxisZ.commands.jogBackward := NOT #TRUE AND "Unit1.Em7.ControlNodes".cm.interlock.sepaGripperAxisZ.permit.jogBackward;
END_REGION

REGION Network 134: CmSepaGripperAxisZ Position Absolute Position0
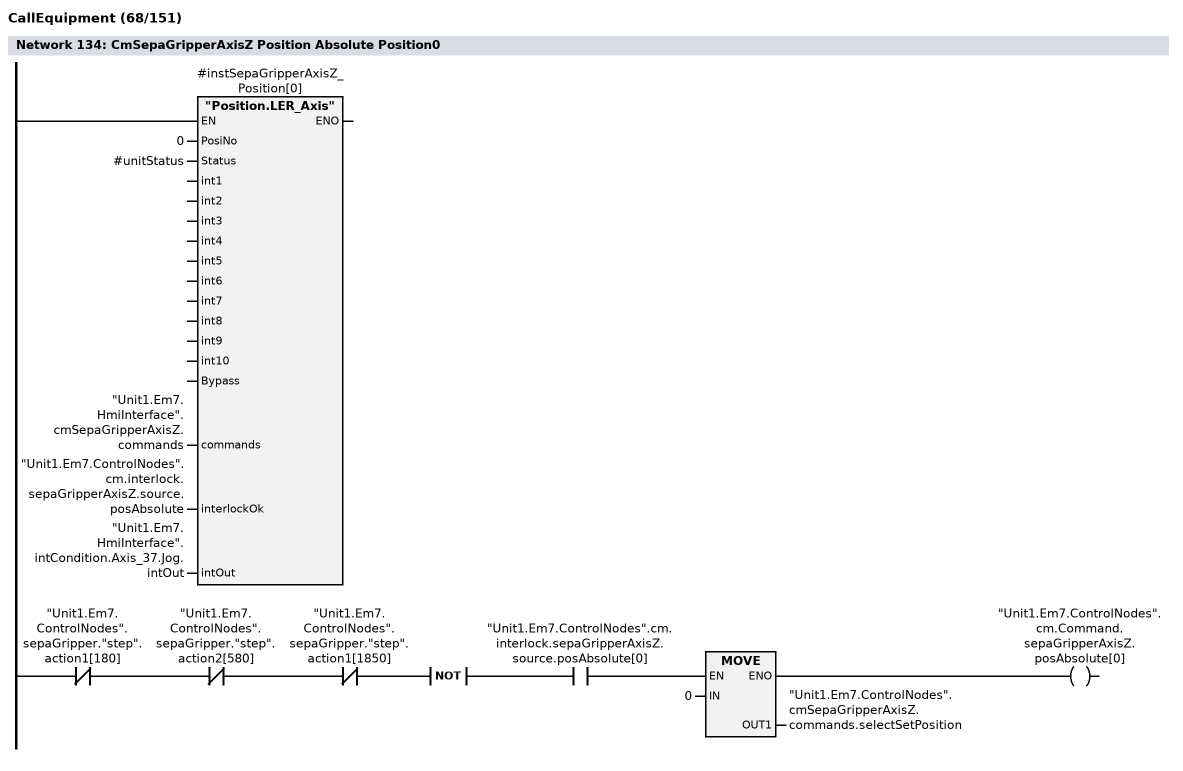
   RUNG wire#powerrail
      #instSepaGripperAxisZ_Position[0](PosiNo := 0, Status := #unitStatus, int1 :=, int2 :=, int3 :=, int4 :=, int5 :=, int6 :=, int7 :=, int8 :=, int9 :=, int10 :=, Bypass :=, commands := "Unit1.Em7.HmiInterface".cmSepaGripperAxisZ.commands, interlockOk := "Unit1.Em7.ControlNodes".cm.interlock.sepaGripperAxisZ.source.posAbsolute, intOut := "Unit1.Em7.HmiInterface".intCondition.Axis_37.Jog.intOut)
   END_RUNG
   RUNG wire#powerrail
      I_Contact( "Unit1.Em7.ControlNodes".sepaGripper."step".action1[180] )
      I_Contact( "Unit1.Em7.ControlNodes".sepaGripper."step".action2[580] )
      I_Contact( "Unit1.Em7.ControlNodes".sepaGripper."step".action1[1850] )
      Not()
      Contact( "Unit1.Em7.ControlNodes".cm.interlock.sepaGripperAxisZ.source.posAbsolute[0] )
      Move(in := 0, out1 => "Unit1.Em7.ControlNodes".cmSepaGripperAxisZ.commands.selectSetPosition)
      Coil( "Unit1.Em7.ControlNodes".cm.Command.sepaGripperAxisZ.posAbsolute[0] )
   END_RUNG
   // the same network as SCL:
   #instSepaGripperAxisZ_Position[0](PosiNo := 0,   // "Position.LER_Axis"
                           Status := #unitStatus,
                           commands := "Unit1.Em7.HmiInterface".cmSepaGripperAxisZ.commands,
                           interlockOk := "Unit1.Em7.ControlNodes".cm.interlock.sepaGripperAxisZ.source.posAbsolute,
                           intOut := "Unit1.Em7.HmiInterface".intCondition.Axis_37.Jog.intOut);
   #_w1 := NOT (NOT "Unit1.Em7.ControlNodes".sepaGripper."step".action1[180] AND NOT "Unit1.Em7.ControlNodes".sepaGripper."step".action2[580] AND NOT "Unit1.Em7.ControlNodes".sepaGripper."step".action1[1850]) AND "Unit1.Em7.ControlNodes".cm.interlock.sepaGripperAxisZ.source.posAbsolute[0];
   IF #_w1 THEN "Unit1.Em7.ControlNodes".cmSepaGripperAxisZ.commands.selectSetPosition := 0; END_IF;
   "Unit1.Em7.ControlNodes".cm.Command.sepaGripperAxisZ.posAbsolute[0] := #_w1;
END_REGION

REGION Network 135: CmSepaGripperAxisZ Position Absolute Position1
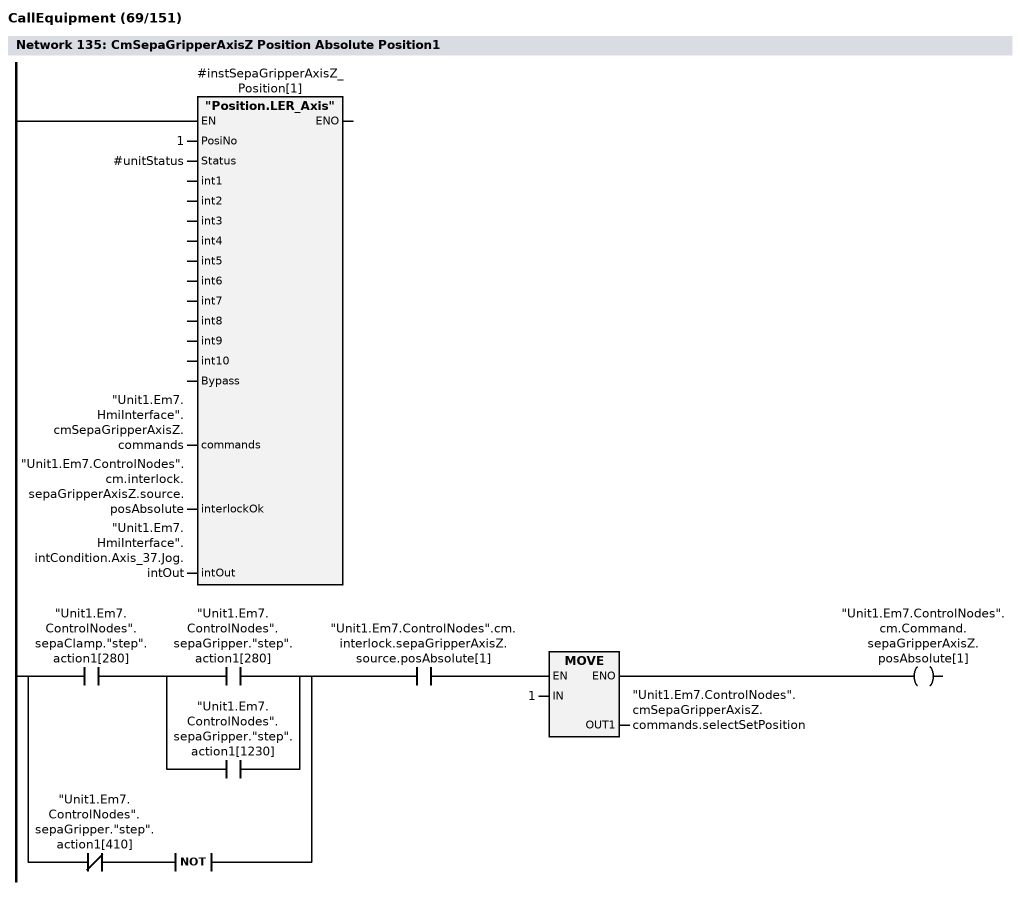
   RUNG wire#powerrail
      #instSepaGripperAxisZ_Position[1](PosiNo := 1, Status := #unitStatus, int1 :=, int2 :=, int3 :=, int4 :=, int5 :=, int6 :=, int7 :=, int8 :=, int9 :=, int10 :=, Bypass :=, commands := "Unit1.Em7.HmiInterface".cmSepaGripperAxisZ.commands, interlockOk := "Unit1.Em7.ControlNodes".cm.interlock.sepaGripperAxisZ.source.posAbsolute, intOut := "Unit1.Em7.HmiInterface".intCondition.Axis_37.Jog.intOut)
   END_RUNG
   RUNG wire#powerrail
      Contact( "Unit1.Em7.ControlNodes".sepaClamp."step".action1[280] )
      wire#w1
      Contact( "Unit1.Em7.ControlNodes".sepaGripper."step".action1[280] )
      wire#w2
      Contact( "Unit1.Em7.ControlNodes".cm.interlock.sepaGripperAxisZ.source.posAbsolute[1] )
      Move(in := 1, out1 => "Unit1.Em7.ControlNodes".cmSepaGripperAxisZ.commands.selectSetPosition)
      Coil( "Unit1.Em7.ControlNodes".cm.Command.sepaGripperAxisZ.posAbsolute[1] )
   END_RUNG
   RUNG wire#w1
      Contact( "Unit1.Em7.ControlNodes".sepaGripper."step".action1[1230] )
   END_RUNG wire#w2
   RUNG wire#powerrail
      I_Contact( "Unit1.Em7.ControlNodes".sepaGripper."step".action1[410] )
      Not()
   END_RUNG wire#w2
   // the same network as SCL:
   #instSepaGripperAxisZ_Position[1](PosiNo := 1,   // "Position.LER_Axis"
                           Status := #unitStatus,
                           commands := "Unit1.Em7.HmiInterface".cmSepaGripperAxisZ.commands,
                           interlockOk := "Unit1.Em7.ControlNodes".cm.interlock.sepaGripperAxisZ.source.posAbsolute,
                           intOut := "Unit1.Em7.HmiInterface".intCondition.Axis_37.Jog.intOut);
   #_w1 := (("Unit1.Em7.ControlNodes".sepaClamp."step".action1[280] AND ("Unit1.Em7.ControlNodes".sepaGripper."step".action1[280] OR "Unit1.Em7.ControlNodes".sepaGripper."step".action1[1230])) OR NOT (NOT "Unit1.Em7.ControlNodes".sepaGripper."step".action1[410])) AND "Unit1.Em7.ControlNodes".cm.interlock.sepaGripperAxisZ.source.posAbsolute[1];
   IF #_w1 THEN "Unit1.Em7.ControlNodes".cmSepaGripperAxisZ.commands.selectSetPosition := 1; END_IF;
   "Unit1.Em7.ControlNodes".cm.Command.sepaGripperAxisZ.posAbsolute[1] := #_w1;
END_REGION

REGION Network 136: CmSepaGripperAxisZ Position Absolute Position2
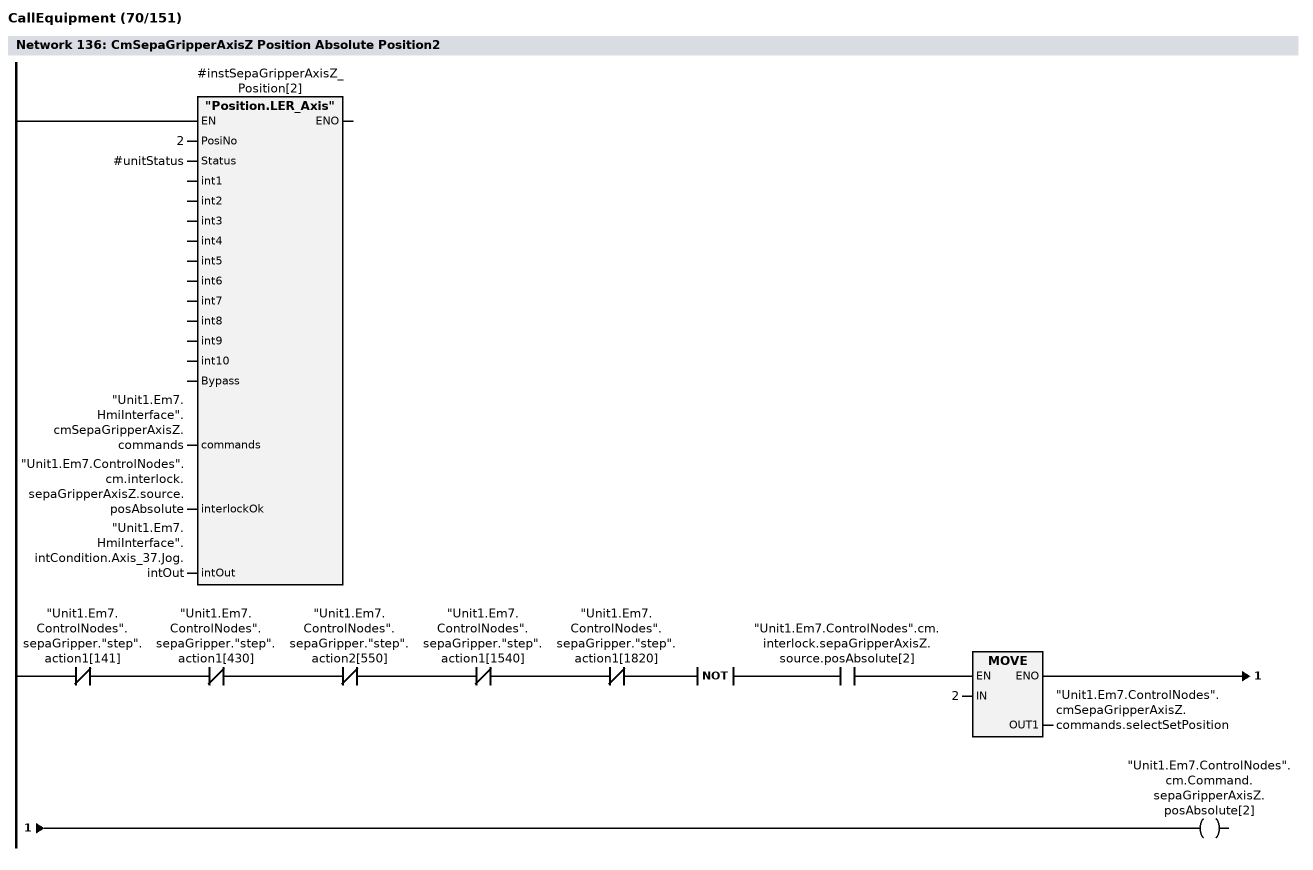
   RUNG wire#powerrail
      #instSepaGripperAxisZ_Position[2](PosiNo := 2, Status := #unitStatus, int1 :=, int2 :=, int3 :=, int4 :=, int5 :=, int6 :=, int7 :=, int8 :=, int9 :=, int10 :=, Bypass :=, commands := "Unit1.Em7.HmiInterface".cmSepaGripperAxisZ.commands, interlockOk := "Unit1.Em7.ControlNodes".cm.interlock.sepaGripperAxisZ.source.posAbsolute, intOut := "Unit1.Em7.HmiInterface".intCondition.Axis_37.Jog.intOut)
   END_RUNG
   RUNG wire#powerrail
      I_Contact( "Unit1.Em7.ControlNodes".sepaGripper."step".action1[141] )
      I_Contact( "Unit1.Em7.ControlNodes".sepaGripper."step".action1[430] )
      I_Contact( "Unit1.Em7.ControlNodes".sepaGripper."step".action2[550] )
      I_Contact( "Unit1.Em7.ControlNodes".sepaGripper."step".action1[1540] )
      I_Contact( "Unit1.Em7.ControlNodes".sepaGripper."step".action1[1820] )
      Not()
      Contact( "Unit1.Em7.ControlNodes".cm.interlock.sepaGripperAxisZ.source.posAbsolute[2] )
      Move(in := 2, out1 => "Unit1.Em7.ControlNodes".cmSepaGripperAxisZ.commands.selectSetPosition)
      Coil( "Unit1.Em7.ControlNodes".cm.Command.sepaGripperAxisZ.posAbsolute[2] )
   END_RUNG
   // the same network as SCL:
   #instSepaGripperAxisZ_Position[2](PosiNo := 2,   // "Position.LER_Axis"
                           Status := #unitStatus,
                           commands := "Unit1.Em7.HmiInterface".cmSepaGripperAxisZ.commands,
                           interlockOk := "Unit1.Em7.ControlNodes".cm.interlock.sepaGripperAxisZ.source.posAbsolute,
                           intOut := "Unit1.Em7.HmiInterface".intCondition.Axis_37.Jog.intOut);
   #_w1 := NOT (NOT "Unit1.Em7.ControlNodes".sepaGripper."step".action1[141] AND NOT "Unit1.Em7.ControlNodes".sepaGripper."step".action1[430] AND NOT "Unit1.Em7.ControlNodes".sepaGripper."step".action2[550] AND NOT "Unit1.Em7.ControlNodes".sepaGripper."step".action1[1540] AND NOT "Unit1.Em7.ControlNodes".sepaGripper."step".action1[1820]) AND "Unit1.Em7.ControlNodes".cm.interlock.sepaGripperAxisZ.source.posAbsolute[2];
   IF #_w1 THEN "Unit1.Em7.ControlNodes".cmSepaGripperAxisZ.commands.selectSetPosition := 2; END_IF;
   "Unit1.Em7.ControlNodes".cm.Command.sepaGripperAxisZ.posAbsolute[2] := #_w1;
END_REGION

REGION Network 137: CmSepaGripperAxisZ Position Absolute Position3
